# B&R Automation Studio project Ampel (part 3)

```cpp
	/// @brief Transition into a state
	///   (if transitioning into a region, activates the state that was active previously)
	/// @param `stateId` State identifier
	HFSM2_CONSTEXPR(14)	void resume   (const StateID stateId_)		noexcept;

	/// @brief Transition into a state
	///   (if transitioning into a region, activates the state that was active previously)
	/// @tparam `TState` State type
	template <typename TState>
	HFSM2_CONSTEXPR(14)	void resume   ()							noexcept	{ resume   (PlanControl::template stateId<TState>());	}

	/// @brief Transition into a state
	///   (if transitioning into a region, activates the sub-state by index returned by the region's `select()` method)
	/// @param `stateId` State identifier
	HFSM2_CONSTEXPR(14)	void select   (const StateID stateId_)		noexcept;

	/// @brief Transition into a state
	///   (if transitioning into a region, activates the sub-state by index returned by the region's `select()` method)
	/// @tparam `TState` State type
	template <typename TState>
	HFSM2_CONSTEXPR(14)	void select   ()							noexcept	{ select   (PlanControl::template stateId<TState>());	}

#if HFSM2_UTILITY_THEORY_AVAILABLE()

	/// @brief Transition into a state
	///   (if transitioning into a region, activates the state with the highest `utility()`
	///   among those with the highest `rank()`)
	/// @param `stateId` State identifier
	/// @see `HFSM2_ENABLE_UTILITY_THEORY`
	HFSM2_CONSTEXPR(14)	void utilize  (const StateID stateId_)		noexcept;

	/// @brief Transition into a state
	///   (if transitioning into a region, activates the state with the highest `utility()`
	///   among those with the highest `rank()`)
	/// @tparam `TState` State type
	/// @see `HFSM2_ENABLE_UTILITY_THEORY`
	template <typename TState>
	HFSM2_CONSTEXPR(14)	void utilize  ()							noexcept	{ utilize  (PlanControl::template stateId<TState>());	}

	/// @brief Transition into a state
	///   (if transitioning into a region, uses weighted random to activate the state proportional to `utility()`
	///   among those with the highest `rank()`)
	/// @param `stateId` State identifier
	/// @see `HFSM2_ENABLE_UTILITY_THEORY`
	HFSM2_CONSTEXPR(14)	void randomize(const StateID stateId_)		noexcept;

	/// @brief Transition into a state
	///   (if transitioning into a region, uses weighted random to activate the state proportional to `utility()`
	///   among those with the highest `rank()`)
	/// @tparam `TState` State type
	/// @see `HFSM2_ENABLE_UTILITY_THEORY`
	template <typename TState>
	HFSM2_CONSTEXPR(14)	void randomize()							noexcept	{ randomize(PlanControl::template stateId<TState>());	}

#endif

	/// @brief Schedule a state to be activated when its parent region is activated
	/// @param `stateId` State identifier
	HFSM2_CONSTEXPR(14)	void schedule (const StateID stateId_)		noexcept;

	/// @brief Schedule a state to be activated when its parent region is activated
	/// @tparam `TState` State type
	template <typename TState>
	HFSM2_CONSTEXPR(14)	void schedule ()							noexcept	{ schedule (PlanControl::template stateId<TState>());	}

#if HFSM2_PLANS_AVAILABLE()

	/// @brief Succeed a plan task for the current state
	/// @see `HFSM2_ENABLE_PLANS`
	HFSM2_CONSTEXPR(14)	void succeed()								noexcept	{ succeed  (_originId							   );	}

	/// @brief Succeed a plan task for a state
	/// @param `stateId` State identifier
	/// @see `HFSM2_ENABLE_PLANS`
	HFSM2_CONSTEXPR(14) void succeed(const StateID stateId_)		noexcept;

	/// @brief Succeed a plan task for a state
	/// @tparam `TState` State type
	/// @see `HFSM2_ENABLE_PLANS`
	template <typename TState>
	HFSM2_CONSTEXPR(14) void succeed()								noexcept	{ succeed  (PlanControl::template stateId<TState>());	}

	/// @brief Fail a plan task for the current state
	/// @see `HFSM2_ENABLE_PLANS`
	HFSM2_CONSTEXPR(14)	void fail	()								noexcept	{ fail	   (_originId							   );	}

	/// @brief Fail a plan task for a state
	/// @param `stateId` State identifier
	/// @see `HFSM2_ENABLE_PLANS`
	HFSM2_CONSTEXPR(14) void fail	(const StateID stateId_)		noexcept;

	/// @brief Fail a plan task for a state
	/// @tparam `TState` State type
	/// @see `HFSM2_ENABLE_PLANS`
	template <typename TState>
	HFSM2_CONSTEXPR(14) void fail	()								noexcept	{ fail	   (PlanControl::template stateId<TState>());	}

#endif

protected:
	using PlanControl::_core;
using PlanControl::_originId;
using PlanControl::_regionId;

using PlanControl::_regionStateId;
using PlanControl::_regionSize;
using PlanControl::_taskStatus;

bool _locked = false;
};

template <typename TArgs>
class FullControlT;

template <
	typename TConfig
  , typename TStateList
  , typename TRegionList
  , Long NCompoCount
  , Long NOrthoCount
  , Long NOrthoUnits
  , typename TReactOrder
  HFSM2_IF_SERIALIZATION(, Long NSerialBits)
  HFSM2_IF_PLANS(, Long NTaskCapacity)
  , typename TPayload
>
class FullControlT<
		  ArgsT<
			  TConfig
			, TStateList
			, TRegionList
			, NCompoCount
			, NOrthoCount
			, NOrthoUnits
			, TReactOrder
			HFSM2_IF_SERIALIZATION(, NSerialBits)
			HFSM2_IF_PLANS(, NTaskCapacity)
			, TPayload
		  >
	  >
	: public FullControlBaseT<
				 ArgsT<
					 TConfig
				   , TStateList
				   , TRegionList
				   , NCompoCount
				   , NOrthoCount
				   , NOrthoUnits
				   , TReactOrder
				   HFSM2_IF_SERIALIZATION(, NSerialBits)
				   HFSM2_IF_PLANS(, NTaskCapacity)
				   , TPayload
				 >
			 >
{
	template <typename, typename, typename>
	friend struct S_;

	template <typename, typename, Strategy, typename, typename...>
	friend struct C_;

	template <typename, typename, typename, typename...>
	friend struct O_;

	template <typename, typename>
	friend class R_;

	using Args = ArgsT<
	TConfig
	, TStateList
	, TRegionList
	, NCompoCount
	, NOrthoCount
	, NOrthoUnits
	, TReactOrder
				   HFSM2_IF_SERIALIZATION(, NSerialBits)
				   HFSM2_IF_PLANS(, NTaskCapacity)
				   , TPayload
				 >;

protected:
	using FullControlBase = FullControlBaseT<Args>;

using typename FullControlBase::Payload;
	using typename FullControlBase::Transition;

	using typename FullControlBase::Origin;

#if HFSM2_PLANS_AVAILABLE()
	using typename FullControlBase::Plan;
	using typename FullControlBase::TasksBits;
#endif

	using FullControlBase::FullControlBase;

#if HFSM2_PLANS_AVAILABLE()

	template <typename TState>
	HFSM2_CONSTEXPR(14)	TaskStatus updatePlan(TState& headState,
											  const TaskStatus subStatus)	noexcept;

#endif

public:
	using FullControlBase::context;

using FullControlBase::isActive;
using FullControlBase::changeTo;

	HFSM2_IF_PLANS(using FullControlBase::plan);

	/// @brief Transition into a state
	///   (if transitioning into a region, acts depending on the region type)
	/// @param `stateId` Destination state identifier
	/// @param `payload` Payload
	HFSM2_CONSTEXPR(14)	void changeWith   (const StateID  stateId_,
										   const Payload& payload)			noexcept;

	/// @brief Transition into a state
	///   (if transitioning into a region, acts depending on the region type)
	/// @tparam `TState` Destination state type
	/// @param `payload` Payload
	template <typename TState>
	HFSM2_CONSTEXPR(14)	void changeWith   (const Payload& payload)			noexcept	{ changeWith   (FullControlBase::template stateId<TState>(),	  payload );	}

	/// @brief Transition into a state
	///   (if transitioning into a region, activates the initial state)
	/// @param `stateId` Destination state identifier
	/// @param `payload` Payload
	HFSM2_CONSTEXPR(14)	void restartWith  (const StateID  stateId_,
										   const Payload& payload)			noexcept;

	/// @brief Transition into a state
	///   (if transitioning into a region, activates the initial state)
	/// @tparam `TState` Destination state type
	/// @param `payload` Payload
	template <typename TState>
	HFSM2_CONSTEXPR(14)	void restartWith  (const Payload& payload)			noexcept	{ restartWith  (FullControlBase::template stateId<TState>(),	  payload );	}

	/// @brief Transition into a state
	///   (if transitioning into a region, activates the state that was active previously)
	/// @param `stateId` Destination state identifier
	/// @param `payload` Payload
	HFSM2_CONSTEXPR(14)	void resumeWith   (const StateID  stateId_,
										   const Payload& payload)			noexcept;

	/// @brief Transition into a state
	///   (if transitioning into a region, activates the state that was active previously)
	/// @tparam `TState` Destination state type
	/// @param `payload` Payload
	template <typename TState>
	HFSM2_CONSTEXPR(14)	void resumeWith   (const Payload& payload)			noexcept	{ resumeWith   (FullControlBase::template stateId<TState>(),	  payload );	}

	/// @brief Transition into a state
	///   (if transitioning into a region, activates the sub-state by index returned by the region's `select()` method)
	/// @param `stateId` Destination state identifier
	/// @param `payload` Payload
	HFSM2_CONSTEXPR(14)	void selectWith   (const StateID  stateId_,
										   const Payload& payload)			noexcept;

	/// @brief Transition into a state
	///   (if transitioning into a region, activates the sub-state by index returned by the region's `select()` method)
	/// @tparam `TState` Destination state type
	/// @param `payload` Payload
	template <typename TState>
	HFSM2_CONSTEXPR(14)	void selectWith   (const Payload& payload)			noexcept	{ selectWith   (FullControlBase::template stateId<TState>(),	  payload );	}

#if HFSM2_UTILITY_THEORY_AVAILABLE()

	/// @brief Transition into a state
	///   (if transitioning into a region, activates the state with the highest `utility()`
	///   among those with the highest `rank()`)
	/// @param `stateId` Destination state identifier
	/// @param `payload` Payload
	/// @see `HFSM2_ENABLE_UTILITY_THEORY`
	HFSM2_CONSTEXPR(14)	void utilizeWith  (const StateID  stateId_,
										   const Payload& payload)			noexcept;

	/// @brief Transition into a state
	///   (if transitioning into a region, activates the state with the highest `utility()`
	///   among those with the highest `rank()`)
	/// @tparam `TState` Destination state type
	/// @param `payload` Payload
	/// @see `HFSM2_ENABLE_UTILITY_THEORY`
	template <typename TState>
	HFSM2_CONSTEXPR(14)	void utilizeWith  (const Payload& payload)			noexcept	{ utilizeWith  (FullControlBase::template stateId<TState>(),	  payload );	}

	/// @brief Transition into a state (if transitioning into a region, uses weighted random to activate the state
	///   proportional to `utility()` among those with the highest `rank()`)
	/// @param `stateId` Destination state identifier
	/// @param `payload` Payload
	/// @see `HFSM2_ENABLE_UTILITY_THEORY`
	HFSM2_CONSTEXPR(14)	void randomizeWith(const StateID  stateId_,
										   const Payload& payload)			noexcept;

	/// @brief Transition into a state (if transitioning into a region, uses weighted random to activate the state
	///   proportional to `utility()` among those with the highest `rank()`)
	/// @tparam `TState` Destination state type
	/// @param `payload` Payload
	/// @see `HFSM2_ENABLE_UTILITY_THEORY`
	template <typename TState>
	HFSM2_CONSTEXPR(14)	void randomizeWith(const Payload& payload)			noexcept	{ randomizeWith(FullControlBase::template stateId<TState>(),	  payload );	}

#endif

	/// @brief Schedule a state to be activated when its parent region is activated
	/// @param `stateId` Destination state identifier
	/// @param `payload` Payload
	HFSM2_CONSTEXPR(14)	void scheduleWith (const StateID  stateId_,
										   const Payload& payload)			noexcept;

	/// @brief Schedule a state to be activated when its parent region is activated
	/// @tparam `TState` Destination state type
	/// @param `payload` Payload
	template <typename TState>
	HFSM2_CONSTEXPR(14)	void scheduleWith (const Payload& payload)			noexcept	{ scheduleWith (FullControlBase::template stateId<TState>(),	  payload );	}

protected:
	using FullControlBase::_core;
using FullControlBase::_originId;
using FullControlBase::_regionId;

using FullControlBase::_regionStateId;
using FullControlBase::_regionSize;
using FullControlBase::_taskStatus;

using FullControlBase::_locked;
};

template <
	typename TConfig
  , typename TStateList
  , typename TRegionList
  , Long NCompoCount
  , Long NOrthoCount
  , Long NOrthoUnits
  , typename TReactOrder
  HFSM2_IF_SERIALIZATION(, Long NSerialBits)
  HFSM2_IF_PLANS(, Long NTaskCapacity)
>
class FullControlT<
		  ArgsT<
			  TConfig
			, TStateList
			, TRegionList
			, NCompoCount
			, NOrthoCount
			, NOrthoUnits
			, TReactOrder
			HFSM2_IF_SERIALIZATION(, NSerialBits)
			HFSM2_IF_PLANS(, NTaskCapacity)
			, void
		  >
	  >
	: public FullControlBaseT<
				 ArgsT<
					 TConfig
				   , TStateList
				   , TRegionList
				   , NCompoCount
				   , NOrthoCount
				   , NOrthoUnits
				   , TReactOrder
				   HFSM2_IF_SERIALIZATION(, NSerialBits)
				   HFSM2_IF_PLANS(, NTaskCapacity)
				   , void
				 >
			 >
{
	template <typename, typename, typename>
	friend struct S_;

	template <typename, typename, Strategy, typename, typename...>
	friend struct C_;

	template <typename, typename, typename, typename...>
	friend struct O_;

	template <typename, typename>
	friend class R_;

	using Args = ArgsT<
	TConfig
	, TStateList
	, TRegionList
	, NCompoCount
	, NOrthoCount
	, NOrthoUnits
	, TReactOrder
				   HFSM2_IF_SERIALIZATION(, NSerialBits)
				   HFSM2_IF_PLANS(, NTaskCapacity)
				   , void
				 >;

protected:
	using FullControlBase = FullControlBaseT<Args>;

using typename FullControlBase::Origin;

#if HFSM2_PLANS_AVAILABLE()
	using typename FullControlBase::Plan;
	using typename FullControlBase::TasksBits;
#endif

	using FullControlBase::FullControlBase;

#if HFSM2_PLANS_AVAILABLE()

	template <typename TState>
	HFSM2_CONSTEXPR(14)	TaskStatus updatePlan(TState& headState,
											  const TaskStatus subStatus)	noexcept;

#endif

public:
	using FullControlBase::context;

using FullControlBase::isActive;
using FullControlBase::changeTo;

	HFSM2_IF_PLANS(using FullControlBase::plan);

protected:
	using FullControlBase::_core;
using FullControlBase::_regionId;

using FullControlBase::_regionStateId;
using FullControlBase::_taskStatus;
};

}
}

namespace hfsm2 {
	namespace detail {

		template <typename TArgs>
		HFSM2_CONSTEXPR(14)
		FullControlBaseT<TArgs>::Lock::Lock(FullControlBaseT& control_) noexcept
	: control{!control_._locked ? &control_ : nullptr}
	{
	if (control)
	control->_locked = true;
}

template <typename TArgs>
HFSM2_CONSTEXPR(20)
FullControlBaseT<TArgs>::Lock::~Lock() noexcept {
	if (control)
control->_locked = false;
}

template <typename TArgs>
HFSM2_CONSTEXPR(14)
void
FullControlBaseT<TArgs>::changeTo(const StateID stateId_) noexcept {
	if (!_locked) {
_core.requests.emplace(Transition{_originId, stateId_, TransitionType::CHANGE});

		if (stateId_ < _regionStateId || _regionStateId + _regionSize <= stateId_)
_taskStatus.outerTransition = true;

		HFSM2_LOG_TRANSITION(context(), _originId, TransitionType::CHANGE, stateId_);
	}
}

template <typename TArgs>
HFSM2_CONSTEXPR(14)
void
FullControlBaseT<TArgs>::restart(const StateID stateId_) noexcept {
	if (!_locked) {
_core.requests.emplace(Transition{_originId, stateId_, TransitionType::RESTART});

		if (stateId_ < _regionStateId || _regionStateId + _regionSize <= stateId_)
_taskStatus.outerTransition = true;

		HFSM2_LOG_TRANSITION(context(), _originId, TransitionType::RESTART, stateId_);
	}
}

template <typename TArgs>
HFSM2_CONSTEXPR(14)
void
FullControlBaseT<TArgs>::resume(const StateID stateId_) noexcept {
	if (!_locked) {
_core.requests.emplace(Transition{_originId, stateId_, TransitionType::RESUME});

		if (stateId_ < _regionStateId || _regionStateId + _regionSize <= stateId_)
_taskStatus.outerTransition = true;

		HFSM2_LOG_TRANSITION(context(), _originId, TransitionType::RESUME, stateId_);
	}
}

template <typename TArgs>
HFSM2_CONSTEXPR(14)
void
FullControlBaseT<TArgs>::select(const StateID stateId_) noexcept {
	if (!_locked) {
_core.requests.emplace(Transition{_originId, stateId_, TransitionType::SELECT});

		if (stateId_ < _regionStateId || _regionStateId + _regionSize <= stateId_)
_taskStatus.outerTransition = true;

		HFSM2_LOG_TRANSITION(context(), _originId, TransitionType::SELECT, stateId_);
	}
}

#if HFSM2_UTILITY_THEORY_AVAILABLE()

template <typename TArgs>
HFSM2_CONSTEXPR(14)
void
FullControlBaseT<TArgs>::utilize(const StateID stateId_) noexcept {
	if (!_locked) {
		_core.requests.emplace(Transition{_originId, stateId_, TransitionType::UTILIZE});

		if (stateId_ < _regionStateId || _regionStateId + _regionSize <= stateId_)
			_taskStatus.outerTransition = true;

		HFSM2_LOG_TRANSITION(context(), _originId, TransitionType::UTILIZE, stateId_);
	}
}

template <typename TArgs>
HFSM2_CONSTEXPR(14)
void
FullControlBaseT<TArgs>::randomize(const StateID stateId_) noexcept {
	if (!_locked) {
_core.requests.emplace(Transition{_originId, stateId_, TransitionType::RANDOMIZE});

		if (stateId_ < _regionStateId || _regionStateId + _regionSize <= stateId_)
_taskStatus.outerTransition = true;

		HFSM2_LOG_TRANSITION(context(), _originId, TransitionType::RANDOMIZE, stateId_);
	}
}

#endif

template <typename TArgs>
HFSM2_CONSTEXPR(14)
void
FullControlBaseT<TArgs>::schedule(const StateID stateId_) noexcept {
_core.requests.emplace(Transition{_originId, stateId_, TransitionType::SCHEDULE});

	HFSM2_LOG_TRANSITION(context(), _originId, TransitionType::SCHEDULE, stateId_);
}

#if HFSM2_PLANS_AVAILABLE()

template <typename TArgs>
HFSM2_CONSTEXPR(14)
void
FullControlBaseT<TArgs>::succeed(const StateID stateId_) noexcept {
	if (ROOT_ID < stateId_ && stateId_ < STATE_COUNT) {
_taskStatus.result = TaskStatus::SUCCESS;

		_core.planData.tasksSuccesses.set(stateId_);

		HFSM2_LOG_TASK_STATUS(context(), _regionStateId, stateId_, StatusEvent::SUCCEEDED);
	}
}

template <typename TArgs>
HFSM2_CONSTEXPR(14)
void
FullControlBaseT<TArgs>::fail(const StateID stateId_) noexcept {
	if (ROOT_ID < stateId_ && stateId_ < STATE_COUNT) {
_taskStatus.result = TaskStatus::FAILURE;

		_core.planData.tasksFailures.set(stateId_);

		HFSM2_LOG_TASK_STATUS(context(), _regionStateId, stateId_, StatusEvent::FAILED);
	}
}

#endif

#if HFSM2_PLANS_AVAILABLE()

template <typename TG_, typename TSL_, typename TRL_, Long NCC_, Long NOC_, Long NOU_, typename TRO_ HFSM2_IF_SERIALIZATION(, Long NSB_), Long NTC_, typename TTP_>
template <typename TState>
HFSM2_CONSTEXPR(14)
TaskStatus
	FullControlT<ArgsT<TG_, TSL_, TRL_, NCC_, NOC_, NOU_, TRO_ HFSM2_IF_SERIALIZATION(, NSB_), NTC_, TTP_>>::updatePlan(TState& headState,
																													const TaskStatus subStatus) noexcept
{
constexpr StateID STATE_ID = TState::STATE_ID; // SPECIFIC

	HFSM2_ASSERT(subStatus);

	if (subStatus.result == TaskStatus::FAILURE) {
_taskStatus.result = TaskStatus::FAILURE;
		HFSM2_LOG_PLAN_STATUS(context(), _regionStateId, StatusEvent::FAILED);

		headState.wrapPlanFailed(*this);

		return TaskStatus{_taskStatus.result};
	} else if (subStatus.result == TaskStatus::SUCCESS) {
if (Plan p = plan(_regionId)) {
TasksBits successesToClear;
			successesToClear.set();

for (auto it = p.begin();
				 it && isActive(it->origin);
				 ++it)
			{
				if (_core.planData.tasksSuccesses.get(it->origin)) {
Origin origin{*this, STATE_ID}; // SPECIFIC

if (const Payload* const payload = it->payload())
						changeWith(it->destination, *it->payload());
					else
						changeTo  (it->destination);

					if (it->cyclic())
						_core.planData.tasksSuccesses.clear(it->origin); // SPECIFIC
					else
						successesToClear.clear(it->origin);

					it.remove();
				}
			}

_core.planData.tasksSuccesses &= successesToClear;

			return TaskStatus{};
		} else {
_taskStatus.result = TaskStatus::SUCCESS;
			HFSM2_LOG_PLAN_STATUS(context(), _regionStateId, StatusEvent::SUCCEEDED);

			plan().clearTasks();
			headState.wrapPlanSucceeded(*this);

			return TaskStatus{_taskStatus.result};
		}
	} else
		return TaskStatus{};
}

#endif

template <typename TG_, typename TSL_, typename TRL_, Long NCC_, Long NOC_, Long NOU_, typename TRO_ HFSM2_IF_SERIALIZATION(, Long NSB_) HFSM2_IF_PLANS(, Long NTC_), typename TTP_>
HFSM2_CONSTEXPR(14)
void
FullControlT<ArgsT<TG_, TSL_, TRL_, NCC_, NOC_, NOU_, TRO_ HFSM2_IF_SERIALIZATION(, NSB_) HFSM2_IF_PLANS(, NTC_), TTP_>>::changeWith(const StateID  stateId_,
																																	 const Payload& payload) noexcept
{
	if (!_locked) {
_core.requests.emplace(Transition{_originId, stateId_, TransitionType::CHANGE, payload});

		if (stateId_ < _regionStateId || _regionStateId + _regionSize <= stateId_)
_taskStatus.outerTransition = true;

		HFSM2_LOG_TRANSITION(context(), _originId, TransitionType::CHANGE, stateId_);
	}
}

template <typename TG_, typename TSL_, typename TRL_, Long NCC_, Long NOC_, Long NOU_, typename TRO_ HFSM2_IF_SERIALIZATION(, Long NSB_) HFSM2_IF_PLANS(, Long NTC_), typename TTP_>
HFSM2_CONSTEXPR(14)
void
FullControlT<ArgsT<TG_, TSL_, TRL_, NCC_, NOC_, NOU_, TRO_ HFSM2_IF_SERIALIZATION(, NSB_) HFSM2_IF_PLANS(, NTC_), TTP_>>::restartWith(const StateID  stateId_,
																																	  const Payload& payload) noexcept
{
	if (!_locked) {
_core.requests.emplace(Transition{_originId, stateId_, TransitionType::RESTART, payload});

		if (stateId_ < _regionStateId || _regionStateId + _regionSize <= stateId_)
_taskStatus.outerTransition = true;

		HFSM2_LOG_TRANSITION(context(), _originId, TransitionType::RESTART, stateId_);
	}
}

template <typename TG_, typename TSL_, typename TRL_, Long NCC_, Long NOC_, Long NOU_, typename TRO_ HFSM2_IF_SERIALIZATION(, Long NSB_) HFSM2_IF_PLANS(, Long NTC_), typename TTP_>
HFSM2_CONSTEXPR(14)
void
FullControlT<ArgsT<TG_, TSL_, TRL_, NCC_, NOC_, NOU_, TRO_ HFSM2_IF_SERIALIZATION(, NSB_) HFSM2_IF_PLANS(, NTC_), TTP_>>::resumeWith(const StateID  stateId_,
																																	 const Payload& payload) noexcept
{
	if (!_locked) {
_core.requests.emplace(Transition{_originId, stateId_, TransitionType::RESUME, payload});

		if (stateId_ < _regionStateId || _regionStateId + _regionSize <= stateId_)
_taskStatus.outerTransition = true;

		HFSM2_LOG_TRANSITION(context(), _originId, TransitionType::RESUME, stateId_);
	}
}

template <typename TG_, typename TSL_, typename TRL_, Long NCC_, Long NOC_, Long NOU_, typename TRO_ HFSM2_IF_SERIALIZATION(, Long NSB_) HFSM2_IF_PLANS(, Long NTC_), typename TTP_>
HFSM2_CONSTEXPR(14)
void
FullControlT<ArgsT<TG_, TSL_, TRL_, NCC_, NOC_, NOU_, TRO_ HFSM2_IF_SERIALIZATION(, NSB_) HFSM2_IF_PLANS(, NTC_), TTP_>>::selectWith(const StateID  stateId_,
																																	 const Payload& payload) noexcept
{
	if (!_locked) {
_core.requests.emplace(Transition{_originId, stateId_, TransitionType::SELECT, payload});

		if (stateId_ < _regionStateId || _regionStateId + _regionSize <= stateId_)
_taskStatus.outerTransition = true;

		HFSM2_LOG_TRANSITION(context(), _originId, TransitionType::SELECT, stateId_);
	}
}

#if HFSM2_UTILITY_THEORY_AVAILABLE()

template <typename TG_, typename TSL_, typename TRL_, Long NCC_, Long NOC_, Long NOU_, typename TRO_ HFSM2_IF_SERIALIZATION(, Long NSB_) HFSM2_IF_PLANS(, Long NTC_), typename TTP_>
HFSM2_CONSTEXPR(14)
void
FullControlT<ArgsT<TG_, TSL_, TRL_, NCC_, NOC_, NOU_, TRO_ HFSM2_IF_SERIALIZATION(, NSB_) HFSM2_IF_PLANS(, NTC_), TTP_>>::utilizeWith(const StateID  stateId_,
																																	  const Payload& payload) noexcept
{
	if (!_locked) {
		_core.requests.emplace(Transition{_originId, stateId_, TransitionType::UTILIZE, payload});

		if (stateId_ < _regionStateId || _regionStateId + _regionSize <= stateId_)
			_taskStatus.outerTransition = true;

		HFSM2_LOG_TRANSITION(context(), _originId, TransitionType::UTILIZE, stateId_);
	}
}

template <typename TG_, typename TSL_, typename TRL_, Long NCC_, Long NOC_, Long NOU_, typename TRO_ HFSM2_IF_SERIALIZATION(, Long NSB_) HFSM2_IF_PLANS(, Long NTC_), typename TTP_>
HFSM2_CONSTEXPR(14)
void
FullControlT<ArgsT<TG_, TSL_, TRL_, NCC_, NOC_, NOU_, TRO_ HFSM2_IF_SERIALIZATION(, NSB_) HFSM2_IF_PLANS(, NTC_), TTP_>>::randomizeWith(const StateID  stateId_,
																																		const Payload& payload) noexcept
{
	if (!_locked) {
		_core.requests.emplace(Transition{_originId, stateId_, TransitionType::RANDOMIZE, payload});

		if (stateId_ < _regionStateId || _regionStateId + _regionSize <= stateId_)
			_taskStatus.outerTransition = true;

		HFSM2_LOG_TRANSITION(context(), _originId, TransitionType::RANDOMIZE, stateId_);
	}
}

#endif

template <typename TG_, typename TSL_, typename TRL_, Long NCC_, Long NOC_, Long NOU_, typename TRO_ HFSM2_IF_SERIALIZATION(, Long NSB_) HFSM2_IF_PLANS(, Long NTC_), typename TTP_>
HFSM2_CONSTEXPR(14)
void
FullControlT<ArgsT<TG_, TSL_, TRL_, NCC_, NOC_, NOU_, TRO_ HFSM2_IF_SERIALIZATION(, NSB_) HFSM2_IF_PLANS(, NTC_), TTP_>>::scheduleWith(const StateID  stateId_,
																																	   const Payload& payload) noexcept
{
_core.requests.emplace(Transition{_originId, stateId_, TransitionType::SCHEDULE, payload});

	HFSM2_LOG_TRANSITION(context(), _originId, TransitionType::SCHEDULE, stateId_);
}

#if HFSM2_PLANS_AVAILABLE()

template <typename TG_, typename TSL_, typename TRL_, Long NCC_, Long NOC_, Long NOU_, typename TRO_ HFSM2_IF_SERIALIZATION(, Long NSB_), Long NTC_>
template <typename TState>
HFSM2_CONSTEXPR(14)
TaskStatus
FullControlT<ArgsT<TG_, TSL_, TRL_, NCC_, NOC_, NOU_, TRO_ HFSM2_IF_SERIALIZATION(, NSB_), NTC_, void>>::updatePlan(TState& headState,
																													const TaskStatus subStatus) noexcept
{
constexpr StateID STATE_ID = TState::STATE_ID; // SPECIFIC

	HFSM2_ASSERT(subStatus);

	if (subStatus.result == TaskStatus::FAILURE) {
_taskStatus.result = TaskStatus::FAILURE;
		HFSM2_LOG_PLAN_STATUS(context(), _regionStateId, StatusEvent::FAILED);

		headState.wrapPlanFailed(*this);

		return TaskStatus{_taskStatus.result};
	} else if (subStatus.result == TaskStatus::SUCCESS) {
if (Plan p = plan(_regionId)) {
TasksBits successesToClear;
			successesToClear.set();

for (auto it = p.begin();
				 it && isActive(it->origin);
				 ++it)
			{
				if (_core.planData.tasksSuccesses.get(it->origin)) {
Origin origin{*this, STATE_ID}; // SPECIFIC

					changeTo(it->destination);

					if (it->cyclic())
						_core.planData.tasksSuccesses.clear(it->origin); // SPECIFIC
					else
						successesToClear.clear(it->origin);

					it.remove();
				}
			}

_core.planData.tasksSuccesses &= successesToClear;

			return TaskStatus{};
		} else {
_taskStatus.result = TaskStatus::SUCCESS;
			HFSM2_LOG_PLAN_STATUS(context(), _regionStateId, StatusEvent::SUCCEEDED);

			plan().clearTasks();
			headState.wrapPlanSucceeded(*this);

			return TaskStatus{_taskStatus.result};
		}
	} else
		return TaskStatus{};
}

#endif

}
}

namespace hfsm2 {
	namespace detail {

		template <typename TArgs>
		class GuardControlT final
		: public FullControlT<TArgs>
		{
		template <typename, typename, typename>
		friend struct S_;

		template <typename, typename>
		friend class R_;

		using FullControl	= FullControlT<TArgs>;

		using typename FullControl::Core;
		using typename FullControl::Context;

		using typename FullControl::Registry;
		using typename FullControl::TransitionSet;
		using typename FullControl::TransitionSets;

#if HFSM2_TRANSITION_HISTORY_AVAILABLE()
		using typename FullControl::TransitionTargets;
#endif

#if HFSM2_UTILITY_THEORY_AVAILABLE()
		using typename FullControl::RNG;
#endif

#if HFSM2_PLANS_AVAILABLE()
		using typename FullControl::PlanData;
#endif

#if HFSM2_LOG_INTERFACE_AVAILABLE()
		using typename FullControl::Logger;
#endif

		HFSM2_CONSTEXPR(11)	GuardControlT(Core& core,
		const TransitionSets& currentTransitions,
		const TransitionSet& pendingTransitions) noexcept
		: FullControl{core, currentTransitions}
, _pendingTransitions{pendingTransitions}
	{}

public:
	using FullControl::context;

	/// @brief Check if a state is going to be activated or deactivated
	/// @param `stateId` State identifier
	/// @return State pending activation/deactivation status
	HFSM2_CONSTEXPR(11)	bool isPendingChange(const StateID stateId_)  const noexcept	{ return _core.registry.isPendingChange(stateId_);					}

	/// @brief Check if a state is going to be activated or deactivated
	/// @tparam `TState` State type
	/// @return State pending activation/deactivation status
	template <typename TState>
	HFSM2_CONSTEXPR(11)	bool isPendingChange()						  const noexcept	{ return isPendingChange(FullControl::template stateId<TState>());	}

	/// @brief Check if a state is going to be activated
	/// @param `stateId` State identifier
	/// @return State pending activation status
	HFSM2_CONSTEXPR(11)	bool isPendingEnter (const StateID stateId_)  const noexcept	{ return _core.registry.isPendingEnter (stateId_);					}

	/// @brief Check if a state is going to be activated
	/// @tparam `TState` State type
	/// @return State pending activation status
	template <typename TState>
	HFSM2_CONSTEXPR(11)	bool isPendingEnter ()						  const noexcept	{ return isPendingEnter (FullControl::template stateId<TState>());	}

	/// @brief Check if a state is going to be deactivated
	/// @param `stateId` State identifier
	/// @return State pending deactivation status
	HFSM2_CONSTEXPR(11)	bool isPendingExit	(const StateID stateId_)  const noexcept	{ return _core.registry.isPendingExit  (stateId_);					}

	/// @brief Check if a state is going to be deactivated
	/// @tparam `TState` State type
	/// @return State pending deactivation status
	template <typename TState>
	HFSM2_CONSTEXPR(11)	bool isPendingExit  ()						  const noexcept	{ return isPendingExit  (FullControl::template stateId<TState>());	}

	/// @brief Get pending transition requests
	/// @return Array of pending transition requests
	HFSM2_CONSTEXPR(11)	const TransitionSet&  pendingTransitions()	  const noexcept	{ return _pendingTransitions;										}

	/// @brief Cancel pending transition requests
	///   (can be used to substitute a transition into the current state with a different one)
	HFSM2_CONSTEXPR(14)	void cancelPendingTransitions()						noexcept;

private:
	using FullControl::_core;
using FullControl::_originId;

const TransitionSet& _pendingTransitions;

bool _cancelled = false;
};

}
}

namespace hfsm2 {
	namespace detail {

		template <typename TArgs>
		HFSM2_CONSTEXPR(14)
		void
		GuardControlT<TArgs>::cancelPendingTransitions() noexcept {
		_cancelled = true;

		HFSM2_LOG_CANCELLED_PENDING(context(), _originId);
	}

}
}

namespace hfsm2 {
	namespace detail {

		template <typename TArgs>
		class EventControlT final
		: public FullControlT<TArgs>
		{
		template <typename, typename>
		friend class R_;

		template <typename, typename>
		friend struct PreReactWrapperT;

		template <typename, typename>
		friend struct ReactWrapperT;

		template <typename, typename>
		friend struct PostReactWrapperT;

		using FullControl	= FullControlT<TArgs>;

		using FullControl::FullControl;

		public:
		using FullControl::context;

		/// @brief Stops processing of the current event down the hierarchy
		/// @see `Config::BottomUpReactions`
	HFSM2_CONSTEXPR(14)	void consumeEvent()								noexcept	{ _consumed = true;	}

	private:
	bool _consumed = false;
};

}
}

namespace hfsm2 {
	namespace detail {

		template <typename TArgs>
		class B_ {
			template <typename...>
			friend struct A_;

			protected:
			using Context		= typename TArgs::Context;

			using Short			= ::hfsm2::Short;
			using Prong			= ::hfsm2::Prong;

#if HFSM2_UTILITY_THEORY_AVAILABLE()
			using Rank			= typename TArgs::Rank;
			using Utility		= typename TArgs::Utility;
#endif

			using StateList		= typename TArgs::StateList;
			using RegionList	= typename TArgs::RegionList;

			using Payload		= typename TArgs::Payload;
			using Transition	= TransitionT<Payload>;

			using ConstControl	= ConstControlT<TArgs>;
			using Control		= ControlT	   <TArgs>;
			using PlanControl	= PlanControlT <TArgs>;
			using FullControl	= FullControlT <TArgs>;
			using GuardControl	= GuardControlT<TArgs>;
			using EventControl	= EventControlT<TArgs>;

#if HFSM2_PLANS_AVAILABLE()
			using Plan			= PayloadPlanT <TArgs>;
#endif

			public:

		HFSM2_CONSTEXPR(14)	void	 entryGuard	  (GuardControl&		 )			noexcept	{}

	HFSM2_CONSTEXPR(14)	void	 enter		  ( PlanControl&		 )			noexcept	{}
HFSM2_CONSTEXPR(14)	void	 reenter	  ( PlanControl&		 )			noexcept	{}

	HFSM2_CONSTEXPR(14)	void	 preUpdate	  ( FullControl&		 )			noexcept	{}
	HFSM2_CONSTEXPR(14)	void	 update		  ( FullControl&		 )			noexcept	{}
	HFSM2_CONSTEXPR(14)	void	 postUpdate	  ( FullControl&		 )			noexcept	{}

	template <typename TEvent>
	HFSM2_CONSTEXPR(14)	void	 preReact	  (const TEvent&		 ,
											   EventControl&		 )			noexcept	{}

	template <typename TEvent>
	HFSM2_CONSTEXPR(14)	void	 react		  (const TEvent&		 ,
											   EventControl&		 )			noexcept	{}

	template <typename TEvent>
	HFSM2_CONSTEXPR(14)	void	 postReact	  (const TEvent&		 ,
											   EventControl&		 )			noexcept	{}

	template <typename TEvent>
	HFSM2_CONSTEXPR(14)	void	 query		  (		 TEvent&		 ,
ConstControl&		 )	  const noexcept	{}

	HFSM2_CONSTEXPR(14)	void	 exitGuard	  (GuardControl&		 )			noexcept	{}

	HFSM2_CONSTEXPR(14)	void	 exit		  ( PlanControl&		 )			noexcept	{}

	template <typename TState>
	static
	HFSM2_CONSTEXPR(11) StateID  stateId()										noexcept	{ return					   index<StateList , TState>() ;	}

	template <typename TState>
	static
	HFSM2_CONSTEXPR(11) RegionID regionId()										noexcept	{ return static_cast<RegionID>(index<RegionList, TState>());	}
};

}
}

namespace hfsm2 {
	namespace detail {

		template <typename...>
		struct A_;

		template <typename TArgs>
		using EmptyT = A_<B_<TArgs>>;

		template <typename TFirst, typename... TRest>
		struct HFSM2_EMPTY_BASES A_<TFirst, TRest...>
		: TFirst
		, A_<TRest...>
		{
		using First		= TFirst;
		using typename First::Context;

#if HFSM2_UTILITY_THEORY_AVAILABLE()
		using typename First::Rank;
		using typename First::Utility;
#endif

		using typename First::StateList;
		using typename First::RegionList;

		using typename First::ConstControl;
		using typename First::Control;
		using typename First::PlanControl;

#if HFSM2_PLANS_AVAILABLE()
		using typename First::Plan;
#endif

		using typename First::FullControl;
		using typename First::GuardControl;
		using typename First::EventControl;

		using First::stateId;
		using First::regionId;

		using Rest		= A_<TRest...>;

		HFSM2_CONSTEXPR(14)	void	 wideEntryGuard(GuardControl& control)			noexcept;

		HFSM2_CONSTEXPR(14)	void	 wideEnter	   ( PlanControl& control)			noexcept;
		HFSM2_CONSTEXPR(14)	void	 wideReenter   ( PlanControl& control)			noexcept;

		HFSM2_CONSTEXPR(14)	void	 widePreUpdate ( FullControl& control)			noexcept;
		HFSM2_CONSTEXPR(14)	void	 wideUpdate	   ( FullControl& control)			noexcept;
		HFSM2_CONSTEXPR(14)	void	 widePostUpdate( FullControl& control)			noexcept;

		template <typename TEvent>
		HFSM2_CONSTEXPR(14)	void	 widePreReact  (const TEvent& event	 ,
		EventControl& control)			noexcept;

		template <typename TEvent>
		HFSM2_CONSTEXPR(14)	void	 wideReact	   (const TEvent& event	 ,
		EventControl& control)			noexcept;

		template <typename TEvent>
		HFSM2_CONSTEXPR(14)	void	 widePostReact (const TEvent& event	 ,
		EventControl& control)			noexcept;

		template <typename TEvent>
		HFSM2_CONSTEXPR(14)	void	 wideQuery	   (	  TEvent& event	 ,
		ConstControl& control)	  const noexcept;

		HFSM2_CONSTEXPR(14)	void	 wideExitGuard (GuardControl& control)			noexcept;

		HFSM2_CONSTEXPR(14)	void	 wideExit	   ( PlanControl& control)			noexcept;

	};

}
}

namespace hfsm2 {
	namespace detail {

		template <typename TF_, typename... TR_>
		HFSM2_CONSTEXPR(14)
		void
		A_<TF_, TR_...>::wideEntryGuard(GuardControl& control) noexcept {
		First::	   entryGuard(control);
		Rest ::wideEntryGuard(control);
	}

	template <typename TF_, typename... TR_>
	HFSM2_CONSTEXPR(14)
	void
	A_<TF_, TR_...>::wideEnter(PlanControl& control) noexcept {
	First::	   enter(control);
	Rest ::wideEnter(control);
}

template <typename TF_, typename... TR_>
HFSM2_CONSTEXPR(14)
void
A_<TF_, TR_...>::wideReenter(PlanControl& control) noexcept {
	First::	   reenter(control);
	Rest ::wideReenter(control);
}

template <typename TF_, typename... TR_>
HFSM2_CONSTEXPR(14)
void
A_<TF_, TR_...>::widePreUpdate(FullControl& control) noexcept {
	First::	   preUpdate(control);
	Rest ::widePreUpdate(control);
}

template <typename TF_, typename... TR_>
HFSM2_CONSTEXPR(14)
void
A_<TF_, TR_...>::wideUpdate(FullControl& control) noexcept {
	First::	   update(control);
	Rest ::wideUpdate(control);
}

template <typename TF_, typename... TR_>
HFSM2_CONSTEXPR(14)
void
A_<TF_, TR_...>::widePostUpdate(FullControl& control) noexcept {
	Rest ::widePostUpdate(control);
	First::	   postUpdate(control);
}

template <typename TF_, typename... TR_>
template <typename TEvent>
HFSM2_CONSTEXPR(14)
void
A_<TF_, TR_...>::widePreReact(const TEvent& event,
							  EventControl& control) noexcept
{
	First::	   preReact(event, control);
	Rest ::widePreReact(event, control);
}

template <typename TF_, typename... TR_>
template <typename TEvent>
HFSM2_CONSTEXPR(14)
void
A_<TF_, TR_...>::wideReact(const TEvent& event,
						   EventControl& control) noexcept
{
	First::	   react(event, control);
	Rest ::wideReact(event, control);
}

template <typename TF_, typename... TR_>
template <typename TEvent>
HFSM2_CONSTEXPR(14)
void
A_<TF_, TR_...>::widePostReact(const TEvent& event,
							   EventControl& control) noexcept
{
	Rest ::widePostReact(event, control);
	First::	   postReact(event, control);
}

template <typename TF_, typename... TR_>
template <typename TEvent>
HFSM2_CONSTEXPR(14)
void
A_<TF_, TR_...>::wideQuery(TEvent& event,
						   ConstControl& control) const noexcept
{
	First::	   query(event, control);
	Rest ::wideQuery(event, control);
}

template <typename TF_, typename... TR_>
HFSM2_CONSTEXPR(14)
void
A_<TF_, TR_...>::wideExitGuard(GuardControl& control) noexcept {
	Rest ::wideExitGuard(control);
	First::	   exitGuard(control);
}

template <typename TF_, typename... TR_>
HFSM2_CONSTEXPR(14)
void
A_<TF_, TR_...>::wideExit(PlanControl& control) noexcept {
	Rest ::wideExit(control);
	First::	   exit(control);
}

}
}

namespace hfsm2 {
	namespace detail {

		template <typename TFirst>
		struct HFSM2_EMPTY_BASES A_<TFirst>
			: TFirst
			{
			using First		= TFirst;
			using typename First::Context;

#if HFSM2_UTILITY_THEORY_AVAILABLE()
			using typename First::Rank;
			using typename First::Utility;
#endif

			using typename First::StateList;
			using typename First::RegionList;

			using typename First::Payload;
			using typename First::Transition;

			using typename First::ConstControl;
			using typename First::Control;
			using typename First::PlanControl;

#if HFSM2_PLANS_AVAILABLE()
			using typename First::Plan;
#endif

			using typename First::FullControl;
			using typename First::GuardControl;
			using typename First::EventControl;

			using First::stateId;
			using First::regionId;

		HFSM2_CONSTEXPR(14)	Prong	 select		   (const Control&		 )			noexcept	{ return 0;					}

#if HFSM2_UTILITY_THEORY_AVAILABLE()
	HFSM2_CONSTEXPR(14)	Rank	 rank		   (const Control&		 )			noexcept	{ return Rank   {0};		}
	HFSM2_CONSTEXPR(14)	Utility  utility	   (const Control&		 )			noexcept	{ return Utility{1};		}
#endif

	HFSM2_CONSTEXPR(14)	void	 entryGuard	   (GuardControl&		 )			noexcept	{}

	HFSM2_CONSTEXPR(14)	void	 enter		   ( PlanControl&		 )			noexcept	{}
	HFSM2_CONSTEXPR(14)	void	 reenter	   ( PlanControl&		 )			noexcept	{}

	HFSM2_CONSTEXPR(14)	void	 preUpdate	   ( FullControl&		 )			noexcept	{}
	HFSM2_CONSTEXPR(14)	void	 update		   ( FullControl&		 )			noexcept	{}
	HFSM2_CONSTEXPR(14)	void	 postUpdate	   ( FullControl&		 )			noexcept	{}

	template <typename TEvent>
	HFSM2_CONSTEXPR(14)	void	 preReact	   (const TEvent&		 ,
												EventControl&		 )			noexcept	{}

	template <typename TEvent>
	HFSM2_CONSTEXPR(14)	void	 react		   (const TEvent&		 ,
												EventControl&		 )			noexcept	{}

	template <typename TEvent>
	HFSM2_CONSTEXPR(14)	void	 postReact	   (const TEvent&		 ,
												EventControl&		 )			noexcept	{}

	template <typename TEvent>
	HFSM2_CONSTEXPR(14)	void	 query		   (	  TEvent&		 ,
ConstControl&		 )	  const noexcept	{}

	HFSM2_CONSTEXPR(14)	void	 exitGuard	   (GuardControl&		 )			noexcept	{}

	HFSM2_CONSTEXPR(14)	void	 exit		   ( PlanControl&		 )			noexcept	{}

#if HFSM2_PLANS_AVAILABLE()
	HFSM2_CONSTEXPR(14)	void	 planSucceeded ( FullControl& control)			noexcept;
	HFSM2_CONSTEXPR(14)	void	 planFailed	   ( FullControl& control)			noexcept;
#endif

	HFSM2_CONSTEXPR(14)	void	 wideEntryGuard(GuardControl& control)			noexcept;

	HFSM2_CONSTEXPR(14)	void	 wideEnter	   ( PlanControl& control)			noexcept;
	HFSM2_CONSTEXPR(14)	void	 wideReenter   ( PlanControl& control)			noexcept;

	HFSM2_CONSTEXPR(14)	void	 widePreUpdate ( FullControl& control)			noexcept;
	HFSM2_CONSTEXPR(14)	void	 wideUpdate	   ( FullControl& control)			noexcept;
	HFSM2_CONSTEXPR(14)	void	 widePostUpdate( FullControl& control)			noexcept;

	template <typename TEvent>
	HFSM2_CONSTEXPR(14)	void	 widePreReact  (const TEvent& event	 ,
												EventControl& control)			noexcept;

	template <typename TEvent>
	HFSM2_CONSTEXPR(14)	void	 wideReact	   (const TEvent& event	 ,
												EventControl& control)			noexcept;

	template <typename TEvent>
	HFSM2_CONSTEXPR(14)	void	 widePostReact (const TEvent& event	 ,
												EventControl& control)			noexcept;

	template <typename TEvent>
	HFSM2_CONSTEXPR(14)	void	 wideQuery	   (	  TEvent& event	 ,
												ConstControl& control)	  const noexcept;

	HFSM2_CONSTEXPR(14)	void	 wideExitGuard (GuardControl& control)			noexcept;

	HFSM2_CONSTEXPR(14)	void	 wideExit	   ( PlanControl& control)			noexcept;

};

}
}

namespace hfsm2 {
	namespace detail {

#if HFSM2_PLANS_AVAILABLE()

		template <typename TF_>
		HFSM2_CONSTEXPR(14)
		void
		A_<TF_>::planSucceeded(FullControl& control) noexcept {
		control.succeed();
	}

	template <typename TF_>
	HFSM2_CONSTEXPR(14)
	void
	A_<TF_>::planFailed(FullControl& control) noexcept {
	control.fail();
}

#endif

template <typename TF_>
HFSM2_CONSTEXPR(14)
void
A_<TF_>::wideEntryGuard(GuardControl& control) noexcept {
	First::	   entryGuard(control);
}

template <typename TF_>
HFSM2_CONSTEXPR(14)
void
A_<TF_>::wideEnter(PlanControl& control) noexcept {
	First::	   enter(control);
}

template <typename TF_>
HFSM2_CONSTEXPR(14)
void
A_<TF_>::wideReenter(PlanControl& control) noexcept {
	First::	   reenter(control);
}

template <typename TF_>
HFSM2_CONSTEXPR(14)
void
A_<TF_>::widePreUpdate(FullControl& control) noexcept {
	First::	   preUpdate(control);
}

template <typename TF_>
HFSM2_CONSTEXPR(14)
void
A_<TF_>::wideUpdate(FullControl& control) noexcept {
	First::	   update(control);
}

template <typename TF_>
HFSM2_CONSTEXPR(14)
void
A_<TF_>::widePostUpdate(FullControl& control) noexcept {
	First::	   postUpdate(control);
}

template <typename TF_>
template <typename TEvent>
HFSM2_CONSTEXPR(14)
void
A_<TF_>::widePreReact(const TEvent& event,
					  EventControl& control) noexcept
{
	First::	   preReact(event, control);
}

template <typename TF_>
template <typename TEvent>
HFSM2_CONSTEXPR(14)
void
A_<TF_>::wideReact(const TEvent& event,
				   EventControl& control) noexcept
{
	First::	   react(event, control);
}

template <typename TF_>
template <typename TEvent>
HFSM2_CONSTEXPR(14)
void
A_<TF_>::widePostReact(const TEvent& event,
					   EventControl& control) noexcept
{
	First::	   postReact(event, control);
}

template <typename TF_>
template <typename TEvent>
HFSM2_CONSTEXPR(14)
void
	A_<TF_>::wideQuery(TEvent& event,
	ConstControl& control) const noexcept
{
	First::	   query(event, control);
}

template <typename TF_>
HFSM2_CONSTEXPR(14)
void
A_<TF_>::wideExitGuard(GuardControl& control) noexcept {
	First::	   exitGuard(control);
}

template <typename TF_>
HFSM2_CONSTEXPR(14)
void
A_<TF_>::wideExit(PlanControl& control) noexcept {
	First::	   exit(control);
}

}
}

namespace hfsm2 {
	namespace detail {

		template <
		typename TIndices
		, typename TArgs
		, typename THead
		>
		struct HFSM2_EMPTY_BASES S_
			: THead
			{
			static constexpr StateID STATE_ID = TIndices::STATE_ID;

			using Context		= typename TArgs::Context;
			using StateList		= typename TArgs::StateList;

#if HFSM2_UTILITY_THEORY_AVAILABLE()
			using Rank			= typename TArgs::Rank;
			using Utility		= typename TArgs::Utility;
			using UP			= typename TArgs::UP;
#endif

#if HFSM2_LOG_INTERFACE_AVAILABLE()
			using Logger		= typename TArgs::Logger;
#endif

			using ConstControl	= ConstControlT<TArgs>;
			using ScopedCOrigin	= typename ConstControl::Origin;

			using Control		= ControlT	   <TArgs>;
			using Registry		= RegistryT	   <TArgs>;
			using StateParents	= typename Registry::StateParents;

			using PlanControl	= PlanControlT <TArgs>;
			using ScopedOrigin	= typename PlanControl::Origin;

			using FullControl	= FullControlT <TArgs>;
			using GuardControl	= GuardControlT<TArgs>;
			using EventControl	= EventControlT<TArgs>;

			using Empty			= EmptyT<TArgs>;
			using Head			= THead;

		HFSM2_CONSTEXPR(14)	Parent		 stateParent		  (		Control& control)								noexcept	{ return control._core.registry.stateParents[STATE_ID];	}

		HFSM2_CONSTEXPR(14)	void		 deepRegister		  (	   Registry& registry, const Parent parent)			noexcept;

		HFSM2_CONSTEXPR(14)	Prong		 wrapSelect			  (		Control& control)								noexcept;

#if HFSM2_UTILITY_THEORY_AVAILABLE()
		HFSM2_CONSTEXPR(14)	Rank		 wrapRank			  (		Control& control)								noexcept;
		HFSM2_CONSTEXPR(14)	Utility		 wrapUtility		  (		Control& control)								noexcept;
#endif

	HFSM2_CONSTEXPR(14)	bool		 deepForwardEntryGuard(GuardControl&		)								noexcept	{ return false;		}
	HFSM2_CONSTEXPR(14)	bool		 deepEntryGuard		  (GuardControl& control)								noexcept;

	HFSM2_CONSTEXPR(14)	void		 deepEnter			  ( PlanControl& control)								noexcept;
	HFSM2_CONSTEXPR(14)	void		 deepReenter		  ( PlanControl& control)								noexcept;

	HFSM2_CONSTEXPR(14)	TaskStatus	 deepPreUpdate		  ( FullControl& control)								noexcept;
	HFSM2_CONSTEXPR(14)	TaskStatus	 deepUpdate			  ( FullControl& control)								noexcept;
	HFSM2_CONSTEXPR(14)	TaskStatus	 deepPostUpdate		  ( FullControl& control)								noexcept;

	template <typename TEvent>
	HFSM2_CONSTEXPR(14)	TaskStatus	 deepPreReact		  (EventControl& control, const TEvent&	event)			noexcept;

	template <typename TEvent>
	HFSM2_CONSTEXPR(14)	TaskStatus	 deepReact			  (EventControl& control, const TEvent&	event)			noexcept;

	template <typename TEvent>
	HFSM2_CONSTEXPR(14)	TaskStatus	 deepPostReact		  (EventControl& control, const TEvent&	event)			noexcept;

	template <typename TEvent>
	HFSM2_CONSTEXPR(14)	void		 deepQuery			  (ConstControl& control,		TEvent& event)	  const noexcept;

#if HFSM2_PLANS_AVAILABLE()
	HFSM2_CONSTEXPR(14)	TaskStatus	 deepUpdatePlans	  ( FullControl& control)								noexcept;
#endif

HFSM2_CONSTEXPR(14)	bool		 deepForwardExitGuard (GuardControl&		)								noexcept	{ return false;		}
	HFSM2_CONSTEXPR(14)	bool		 deepExitGuard		  (GuardControl& control)								noexcept;

	HFSM2_CONSTEXPR(14)	void		 deepExit			  ( PlanControl& control)								noexcept;

#if HFSM2_PLANS_AVAILABLE()
	HFSM2_CONSTEXPR(14)	void		 wrapPlanSucceeded	  ( FullControl& control)								noexcept;
	HFSM2_CONSTEXPR(14)	void		 wrapPlanFailed		  ( FullControl& control)								noexcept;
#endif

	HFSM2_CONSTEXPR(14)	void		 deepForwardActive	  (	    Control&,		  const Request		   )		noexcept	{}
	HFSM2_CONSTEXPR(14)	void		 deepForwardRequest	  (	    Control& control, const Request request)		noexcept;

	HFSM2_CONSTEXPR(14)	void		 deepRequestChange	  (	    Control& control, const Request request)		noexcept;
	HFSM2_CONSTEXPR(14)	void		 deepRequestRestart	  (		Control& control, const Request request)		noexcept;
	HFSM2_CONSTEXPR(14)	void		 deepRequestResume	  (		Control& control, const Request request)		noexcept;
	HFSM2_CONSTEXPR(14)	void		 deepRequestSelect	  (	    Control& control, const Request request)		noexcept;

#if HFSM2_UTILITY_THEORY_AVAILABLE()
	HFSM2_CONSTEXPR(14)	void		 deepRequestUtilize	  (		Control& control, const Request request)		noexcept;
	HFSM2_CONSTEXPR(14)	void		 deepRequestRandomize (		Control& control, const Request request)		noexcept;

	HFSM2_CONSTEXPR(14)	UP			 deepReportChange	  (	    Control& control)								noexcept;
	HFSM2_CONSTEXPR(14)	UP			 deepReportUtilize	  (	    Control& control)								noexcept;
	HFSM2_CONSTEXPR(14)	Rank		 deepReportRank		  (		Control& control)								noexcept;
	HFSM2_CONSTEXPR(14)	Utility		 deepReportRandomize  (	    Control& control)								noexcept;
#endif

	HFSM2_CONSTEXPR(14)	void		 deepChangeToRequested(	   Control&)										noexcept	{}

#if HFSM2_SERIALIZATION_AVAILABLE()
	using WriteStream	= typename TArgs::WriteStream;
	using ReadStream	= typename TArgs::ReadStream;

	HFSM2_CONSTEXPR(14)	void		 deepSaveActive		  (const Registry&, WriteStream&)				  const noexcept	{}
	HFSM2_CONSTEXPR(14)	void		 deepSaveResumable	  (const Registry&, WriteStream&)				  const noexcept	{}

	HFSM2_CONSTEXPR(14)	void		 deepLoadRequested	  (		 Registry&,  ReadStream&)				  const noexcept	{}
	HFSM2_CONSTEXPR(14)	void		 deepLoadResumable	  (		 Registry&,  ReadStream&)				  const noexcept	{}
#endif

#if HFSM2_STRUCTURE_REPORT_AVAILABLE()
	using StructureStateInfos = typename TArgs::StructureStateInfos;

	static
	HFSM2_CONSTEXPR(NO)	const char* name() noexcept;

	HFSM2_CONSTEXPR(14)	void deepGetNames(const Long parent,
										  const RegionType region,
										  const Short depth,
										  StructureStateInfos& stateInfos)							  const noexcept;
#endif

#if HFSM2_DEBUG_STATE_TYPE_AVAILABLE() || HFSM2_STRUCTURE_REPORT_AVAILABLE() || HFSM2_LOG_INTERFACE_AVAILABLE()

	HFSM2_IF_TYPEINDEX(const std::type_index TYPE = typeid(Head));

	static constexpr Long NAME_COUNT = 1;

#endif

#if HFSM2_LOG_INTERFACE_AVAILABLE()

	template <typename TReturn, typename THost, typename... TParams>
	HFSM2_CONSTEXPR(14)
	void log(TReturn (THost::*)(TParams...),
Logger& logger,
const Context& context,
const Method method)																	  const noexcept
	{
		logger.recordMethod(context, STATE_ID, method);
	}

	template <typename TReturn, typename THost, typename... TParams>
	HFSM2_CONSTEXPR(14)
	void log(TReturn (THost::*)(TParams...) const,
Logger& logger,
const Context& context,
const Method method)																	  const noexcept
	{
		logger.recordMethod(context, STATE_ID, method);
	}

	template <typename TReturn, typename... TParams>
	HFSM2_CONSTEXPR(14)
	void log(TReturn (Empty::*)(TParams...),
Logger&,
const Context&,
			 const Method)																			  const noexcept
	{}

	template <typename TReturn, typename... TParams>
	HFSM2_CONSTEXPR(14)
	void log(TReturn (Empty::*)(TParams...) const,
Logger&,
const Context&,
			 const Method)																			  const noexcept
	{}

#endif
};

}
}

namespace hfsm2 {
	namespace detail {

		template <typename TN_, typename TA_, typename TH_>
		HFSM2_CONSTEXPR(14)
		void
		S_<TN_, TA_, TH_>::deepRegister(Registry& registry,
		const Parent parent) noexcept
		{
		constexpr StateID HEAD_ID = index<StateList, TH_>();
		static_assert(STATE_ID == HEAD_ID, "");

		registry.stateParents[STATE_ID] = parent;
	}

	template <typename TN_, typename TA_, typename TH_>
	HFSM2_CONSTEXPR(14)
	Prong
	S_<TN_, TA_, TH_>::wrapSelect(Control& control) noexcept {
	HFSM2_LOG_STATE_METHOD(&Head::select,
	Method::SELECT);

	return Head::select(static_cast<const Control&>(control));
}

#if HFSM2_UTILITY_THEORY_AVAILABLE()

template <typename TN_, typename TA_, typename TH_>
HFSM2_CONSTEXPR(14)
typename S_<TN_, TA_, TH_>::Rank
S_<TN_, TA_, TH_>::wrapRank(Control& control) noexcept {
	HFSM2_LOG_STATE_METHOD(&Head::rank,
						   Method::RANK);

	return Head::rank(static_cast<const Control&>(control));
}

template <typename TN_, typename TA_, typename TH_>
HFSM2_CONSTEXPR(14)
typename S_<TN_, TA_, TH_>::Utility
S_<TN_, TA_, TH_>::wrapUtility(Control& control) noexcept {
	HFSM2_LOG_STATE_METHOD(&Head::utility,
						   Method::UTILITY);

	return Head::utility(static_cast<const Control&>(control));
}

#endif

template <typename TN_, typename TA_, typename TH_>
HFSM2_CONSTEXPR(14)
bool
S_<TN_, TA_, TH_>::deepEntryGuard(GuardControl& control) noexcept {
	HFSM2_LOG_STATE_METHOD(&Head::entryGuard,
						   Method::ENTRY_GUARD);

ScopedOrigin origin{control, STATE_ID};

const bool cancelledBefore = control._cancelled;

	Head::wideEntryGuard(control);
	Head::	  entryGuard(control);

return !cancelledBefore && control._cancelled;
}

template <typename TN_, typename TA_, typename TH_>
HFSM2_CONSTEXPR(14)
void
S_<TN_, TA_, TH_>::deepEnter(PlanControl& control) noexcept {
	HFSM2_IF_PLANS(control._core.planData.verifyEmptyStatus(STATE_ID));

	HFSM2_LOG_STATE_METHOD(&Head::enter,
						   Method::ENTER);

ScopedOrigin origin{control, STATE_ID};

	Head::wideEnter(control);
	Head::	  enter(control);
}

template <typename TN_, typename TA_, typename TH_>
HFSM2_CONSTEXPR(14)
void
S_<TN_, TA_, TH_>::deepReenter(PlanControl& control) noexcept {
	HFSM2_IF_PLANS(control._core.planData.verifyEmptyStatus(STATE_ID));

	HFSM2_LOG_STATE_METHOD(&Head::reenter,
						   Method::REENTER);

ScopedOrigin origin{control, STATE_ID};

	Head::wideReenter(control);
	Head::	  reenter(control);
}

template <typename TN_, typename TA_, typename TH_>
HFSM2_CONSTEXPR(14)
TaskStatus
S_<TN_, TA_, TH_>::deepPreUpdate(FullControl& control) noexcept {
	HFSM2_LOG_STATE_METHOD(&Head::preUpdate,
						   Method::PRE_UPDATE);

ScopedOrigin origin{control, STATE_ID};

	Head::widePreUpdate(control);
	Head::	  preUpdate(control);

return control._taskStatus;
}

template <typename TN_, typename TA_, typename TH_>
HFSM2_CONSTEXPR(14)
TaskStatus
S_<TN_, TA_, TH_>::deepUpdate(FullControl& control) noexcept {
	HFSM2_LOG_STATE_METHOD(&Head::update,
						   Method::UPDATE);

ScopedOrigin origin{control, STATE_ID};

	Head::wideUpdate(control);
	Head::	  update(control);

return control._taskStatus;
}

template <typename TN_, typename TA_, typename TH_>
HFSM2_CONSTEXPR(14)
TaskStatus
S_<TN_, TA_, TH_>::deepPostUpdate(FullControl& control) noexcept {
	HFSM2_LOG_STATE_METHOD(&Head::postUpdate,
						   Method::POST_UPDATE);

ScopedOrigin origin{control, STATE_ID};

	Head::	  postUpdate(control);
	Head::widePostUpdate(control);

return control._taskStatus;
}

template <typename TN_, typename TA_, typename TH_>
template <typename TEvent>
HFSM2_CONSTEXPR(14)
TaskStatus
S_<TN_, TA_, TH_>::deepPreReact(EventControl& control,
								const TEvent& event) noexcept
{
auto method = static_cast<void (Head::*)(const TEvent&, EventControl&)>(&Head::preReact);

	HFSM2_LOG_STATE_METHOD(method,
						   Method::PRE_REACT);

ScopedOrigin origin{control, STATE_ID};

	Head::widePreReact(event, control);
(this->*method) (event, control);

return control._taskStatus;
}

template <typename TN_, typename TA_, typename TH_>
template <typename TEvent>
HFSM2_CONSTEXPR(14)
TaskStatus
S_<TN_, TA_, TH_>::deepReact(EventControl& control,
							 const TEvent& event) noexcept
{
auto method = static_cast<void (Head::*)(const TEvent&, EventControl&)>(&Head::react);

	HFSM2_LOG_STATE_METHOD(method,
						   Method::REACT);

ScopedOrigin origin{control, STATE_ID};

	Head::wideReact(event, control);
(this->*method)(event, control);

return control._taskStatus;
}

template <typename TN_, typename TA_, typename TH_>
template <typename TEvent>
HFSM2_CONSTEXPR(14)
TaskStatus
S_<TN_, TA_, TH_>::deepPostReact(EventControl& control,
								 const TEvent& event) noexcept
{
auto method = static_cast<void (Head::*)(const TEvent&, EventControl&)>(&Head::postReact);

	HFSM2_LOG_STATE_METHOD(method,
						   Method::POST_REACT);

ScopedOrigin origin{control, STATE_ID};

(this->*method)	   (event, control);
	Head::widePostReact(event, control);

return control._taskStatus;
}

template <typename TN_, typename TA_, typename TH_>
template <typename TEvent>
HFSM2_CONSTEXPR(14)
void
	S_<TN_, TA_, TH_>::deepQuery(ConstControl& control,
	TEvent&  event) const noexcept
{
	auto method = static_cast<void (Head::*)(TEvent&, ConstControl&) const>(&Head::query);

	HFSM2_LOG_STATE_METHOD(method,
		Method::QUERY);

	ScopedCOrigin origin{control, STATE_ID};

	(this->*method)(event, control);
		Head::wideQuery(event, control);
}

#if HFSM2_PLANS_AVAILABLE()

template <typename TN_, typename TA_, typename TH_>
HFSM2_CONSTEXPR(14)
TaskStatus
S_<TN_, TA_, TH_>::deepUpdatePlans(FullControl& control) noexcept {
	if (control._core.planData.tasksFailures .get(STATE_ID))
		return TaskStatus{TaskStatus::FAILURE};
	else
	if (control._core.planData.tasksSuccesses.get(STATE_ID))
		return TaskStatus{TaskStatus::SUCCESS};
	else
		return TaskStatus{};
}

#endif

template <typename TN_, typename TA_, typename TH_>
HFSM2_CONSTEXPR(14)
bool
S_<TN_, TA_, TH_>::deepExitGuard(GuardControl& control) noexcept {
	HFSM2_LOG_STATE_METHOD(&Head::exitGuard,
						   Method::EXIT_GUARD);

ScopedOrigin origin{control, STATE_ID};

const bool cancelledBefore = control._cancelled;

	Head::wideExitGuard(control);
	Head::	  exitGuard(control);

return !cancelledBefore && control._cancelled;
}

template <typename TN_, typename TA_, typename TH_>
HFSM2_CONSTEXPR(14)
void
S_<TN_, TA_, TH_>::deepExit(PlanControl& control) noexcept {
	HFSM2_LOG_STATE_METHOD(&Head::exit,
						   Method::EXIT);

ScopedOrigin origin{control, STATE_ID};

	// if you see..
	// VS	 - error C2039:  'exit': is not a member of 'Blah'
	// Clang - error : no member named 'exit' in 'Blah'
	//
	// .. inherit state 'Blah' from hfsm2::Machine::Instance::State
	Head::	  exit(control);
	Head::wideExit(control);

	HFSM2_IF_PLANS(control._core.planData.clearTaskStatus(STATE_ID));
}

#if HFSM2_PLANS_AVAILABLE()

template <typename TN_, typename TA_, typename TH_>
HFSM2_CONSTEXPR(14)
void
S_<TN_, TA_, TH_>::wrapPlanSucceeded(FullControl& control) noexcept {
	HFSM2_LOG_STATE_METHOD(&Head::planSucceeded,
						   Method::PLAN_SUCCEEDED);

ScopedOrigin origin{control, STATE_ID};

	Head::planSucceeded(control);
}

template <typename TN_, typename TA_, typename TH_>
HFSM2_CONSTEXPR(14)
void
S_<TN_, TA_, TH_>::wrapPlanFailed(FullControl& control) noexcept {
	HFSM2_LOG_STATE_METHOD(&Head::planFailed,
						   Method::PLAN_FAILED);

ScopedOrigin origin{control, STATE_ID};

	Head::planFailed(control);
}

#endif

template <typename TN_, typename TA_, typename TH_>
HFSM2_CONSTEXPR(14)
void
S_<TN_, TA_, TH_>::deepForwardRequest(Control& HFSM2_IF_TRANSITION_HISTORY(control),
									  const Request HFSM2_IF_TRANSITION_HISTORY(request)) noexcept
{
	HFSM2_IF_TRANSITION_HISTORY(control.pinLastTransition(STATE_ID, request.index));
}

template <typename TN_, typename TA_, typename TH_>
HFSM2_CONSTEXPR(14)
void
S_<TN_, TA_, TH_>::deepRequestChange(Control& HFSM2_IF_TRANSITION_HISTORY(control),
									 const Request HFSM2_IF_TRANSITION_HISTORY(request)) noexcept
{
	HFSM2_IF_TRANSITION_HISTORY(control.pinLastTransition(STATE_ID, request.index));
}

template <typename TN_, typename TA_, typename TH_>
HFSM2_CONSTEXPR(14)
void
S_<TN_, TA_, TH_>::deepRequestRestart(Control& HFSM2_IF_TRANSITION_HISTORY(control),
									  const Request HFSM2_IF_TRANSITION_HISTORY(request)) noexcept
{
	HFSM2_IF_TRANSITION_HISTORY(control.pinLastTransition(STATE_ID, request.index));
}

template <typename TN_, typename TA_, typename TH_>
HFSM2_CONSTEXPR(14)
void
S_<TN_, TA_, TH_>::deepRequestResume(Control& HFSM2_IF_TRANSITION_HISTORY(control),
									 const Request HFSM2_IF_TRANSITION_HISTORY(request)) noexcept
{
	HFSM2_IF_TRANSITION_HISTORY(control.pinLastTransition(STATE_ID, request.index));
}

template <typename TN_, typename TA_, typename TH_>
HFSM2_CONSTEXPR(14)
void
S_<TN_, TA_, TH_>::deepRequestSelect(Control& HFSM2_IF_TRANSITION_HISTORY(control),
									 const Request HFSM2_IF_TRANSITION_HISTORY(request)) noexcept
{
	HFSM2_IF_TRANSITION_HISTORY(control.pinLastTransition(STATE_ID, request.index));
}

#if HFSM2_UTILITY_THEORY_AVAILABLE()

template <typename TN_, typename TA_, typename TH_>
HFSM2_CONSTEXPR(14)
void
S_<TN_, TA_, TH_>::deepRequestUtilize(Control& HFSM2_IF_TRANSITION_HISTORY(control),
									  const Request HFSM2_IF_TRANSITION_HISTORY(request)) noexcept
{
	HFSM2_IF_TRANSITION_HISTORY(control.pinLastTransition(STATE_ID, request.index));
}

template <typename TN_, typename TA_, typename TH_>
HFSM2_CONSTEXPR(14)
void
S_<TN_, TA_, TH_>::deepRequestRandomize(Control& HFSM2_IF_TRANSITION_HISTORY(control),
										const Request HFSM2_IF_TRANSITION_HISTORY(request)) noexcept
{
	HFSM2_IF_TRANSITION_HISTORY(control.pinLastTransition(STATE_ID, request.index));
}

template <typename TN_, typename TA_, typename TH_>
HFSM2_CONSTEXPR(14)
typename S_<TN_, TA_, TH_>::UP
S_<TN_, TA_, TH_>::deepReportChange(Control& control) noexcept {
const Utility utility = wrapUtility(control);

const Parent parent = stateParent(control);

return {utility, parent.prong};
}

template <typename TN_, typename TA_, typename TH_>
HFSM2_CONSTEXPR(14)
typename S_<TN_, TA_, TH_>::UP
S_<TN_, TA_, TH_>::deepReportUtilize(Control& control) noexcept {
const Utility utility = wrapUtility(control);
const Parent  parent  = stateParent(control);

return {utility, parent.prong};
}

template <typename TN_, typename TA_, typename TH_>
HFSM2_CONSTEXPR(14)
typename S_<TN_, TA_, TH_>::Rank
S_<TN_, TA_, TH_>::deepReportRank(Control& control) noexcept {
	return wrapRank(control);
}

template <typename TN_, typename TA_, typename TH_>
HFSM2_CONSTEXPR(14)
typename S_<TN_, TA_, TH_>::Utility
S_<TN_, TA_, TH_>::deepReportRandomize(Control& control) noexcept {
	return wrapUtility(control);
}

#endif

#if HFSM2_STRUCTURE_REPORT_AVAILABLE()

template <typename TN_, typename TA_, typename TH_>
HFSM2_CONSTEXPR(NO)
const char*
S_<TN_, TA_, TH_>::name() noexcept {
const std::type_index type = typeid(Head);
const char* const raw = type.name();

#if defined(_MSC_VER)

	Short first =
		raw[0] == 's' ? 7 : // Struct
		raw[0] == 'c' ? 6 : // Class
						0;

for (Short c = first; raw[c]; ++c)
if (raw[c] == ':')
first = c + 1;

return raw + first;

#elif defined(__clang__) || defined(__GNUC__) || defined(__GNUG__)

return raw;

#else

return raw;

#endif
}

template <typename TN_, typename TA_, typename TH_>
HFSM2_CONSTEXPR(14)
void
	S_<TN_, TA_, TH_>::deepGetNames(const Long parent,
	const RegionType region,
	const Short depth,
	StructureStateInfos& stateInfos) const noexcept
{
	stateInfos.emplace(StructureStateInfo{parent, region, depth, name()});
		}

#endif

}
}

namespace hfsm2 {
	namespace detail {

#if HFSM2_DEBUG_STATE_TYPE_AVAILABLE() || HFSM2_STRUCTURE_REPORT_AVAILABLE() || HFSM2_LOG_INTERFACE_AVAILABLE()

		struct None final {};

#endif

	template <
	typename TIndices
	, typename TArgs
	>
	struct S_<TIndices, TArgs, EmptyT<TArgs>>
		: EmptyT<TArgs>
		{
		static constexpr StateID STATE_ID = TIndices::STATE_ID;

		using Context		= typename TArgs::Context;

#if HFSM2_UTILITY_THEORY_AVAILABLE()
		using Rank			= typename TArgs::Rank;
		using Utility		= typename TArgs::Utility;
		using UP			= typename TArgs::UP;
#endif

#if HFSM2_LOG_INTERFACE_AVAILABLE()
		using Logger		= typename TArgs::Logger;
#endif

		using ConstControl	= ConstControlT<TArgs>;
		using ScopedCOrigin	= typename ConstControl::Origin;

		using Control		= ControlT	   <TArgs>;
		using Registry		= RegistryT	   <TArgs>;
		using StateParents	= typename Registry::StateParents;

		using PlanControl	= PlanControlT <TArgs>;
		using ScopedOrigin	= typename PlanControl::Origin;

		using FullControl	= FullControlT <TArgs>;
		using GuardControl	= GuardControlT<TArgs>;
		using EventControl	= EventControlT<TArgs>;

		using Empty			= EmptyT<TArgs>;
		using Head			= Empty;

	HFSM2_CONSTEXPR(14)	Parent		 stateParent		  (		Control& control)								noexcept	{ return control._core.registry.stateParents[STATE_ID];	}

	HFSM2_CONSTEXPR(14)	void		 deepRegister		  (	   Registry& registry, const Parent parent)			noexcept;

	HFSM2_CONSTEXPR(14)	Prong		 wrapSelect			  (		Control& control)								noexcept;

#if HFSM2_UTILITY_THEORY_AVAILABLE()
	HFSM2_CONSTEXPR(14)	Rank		 wrapRank			  (		Control& control)								noexcept;
	HFSM2_CONSTEXPR(14)	Utility		 wrapUtility		  (		Control& control)								noexcept;
#endif

HFSM2_CONSTEXPR(14)	bool		 deepForwardEntryGuard(GuardControl&		)								noexcept	{ return false;		}
	HFSM2_CONSTEXPR(14)	bool		 deepEntryGuard		  (GuardControl& control)								noexcept;

	HFSM2_CONSTEXPR(14)	void		 deepEnter			  ( PlanControl& control)								noexcept;
	HFSM2_CONSTEXPR(14)	void		 deepReenter		  ( PlanControl& control)								noexcept;

	HFSM2_CONSTEXPR(14)	TaskStatus	 deepPreUpdate		  ( FullControl& control)								noexcept;
	HFSM2_CONSTEXPR(14)	TaskStatus	 deepUpdate			  ( FullControl& control)								noexcept;
	HFSM2_CONSTEXPR(14)	TaskStatus	 deepPostUpdate		  ( FullControl& control)								noexcept;

	template <typename TEvent>
	HFSM2_CONSTEXPR(14)	TaskStatus	 deepPreReact		  (EventControl& control, const TEvent&	event)			noexcept;

	template <typename TEvent>
	HFSM2_CONSTEXPR(14)	TaskStatus	 deepReact			  (EventControl& control, const TEvent&	event)			noexcept;

	template <typename TEvent>
	HFSM2_CONSTEXPR(14)	TaskStatus	 deepPostReact		  (EventControl& control, const TEvent&	event)			noexcept;

	template <typename TEvent>
	HFSM2_CONSTEXPR(14)	void		 deepQuery			  (ConstControl& control,		TEvent& event)	  const noexcept;

#if HFSM2_PLANS_AVAILABLE()
	HFSM2_CONSTEXPR(14)	TaskStatus	 deepUpdatePlans	  ( FullControl& control)								noexcept;
#endif

	HFSM2_CONSTEXPR(14)	bool		 deepForwardExitGuard (GuardControl&		)								noexcept	{ return false;		}
	HFSM2_CONSTEXPR(14)	bool		 deepExitGuard		  (GuardControl& control)								noexcept;

	HFSM2_CONSTEXPR(14)	void		 deepExit			  ( PlanControl& control)								noexcept;

#if HFSM2_PLANS_AVAILABLE()
	HFSM2_CONSTEXPR(14)	void		 wrapPlanSucceeded	  ( FullControl& control)								noexcept;
	HFSM2_CONSTEXPR(14)	void		 wrapPlanFailed		  ( FullControl& control)								noexcept;
#endif

	HFSM2_CONSTEXPR(14)	void		 deepForwardActive	  (	   Control&,		 const Request		  )			noexcept	{}
	HFSM2_CONSTEXPR(14)	void		 deepForwardRequest	  (	   Control& control, const Request request)			noexcept;

	HFSM2_CONSTEXPR(14)	void		 deepRequestChange	  (	    Control& control, const Request request)		noexcept;
	HFSM2_CONSTEXPR(14)	void		 deepRequestRestart	  (		Control& control, const Request request)		noexcept;
	HFSM2_CONSTEXPR(14)	void		 deepRequestResume	  (		Control& control, const Request request)		noexcept;
	HFSM2_CONSTEXPR(14)	void		 deepRequestSelect	  (	    Control& control, const Request request)		noexcept;

#if HFSM2_UTILITY_THEORY_AVAILABLE()
	HFSM2_CONSTEXPR(14)	void		 deepRequestUtilize	  (		Control& control, const Request request)		noexcept;
	HFSM2_CONSTEXPR(14)	void		 deepRequestRandomize (		Control& control, const Request request)		noexcept;

	HFSM2_CONSTEXPR(14)	UP			 deepReportChange	  (	    Control& control)								noexcept;
	HFSM2_CONSTEXPR(14)	UP			 deepReportUtilize	  (	    Control& control)								noexcept;
	HFSM2_CONSTEXPR(14)	Rank		 deepReportRank		  (		Control& control)								noexcept;
	HFSM2_CONSTEXPR(14)	Utility		 deepReportRandomize  (	    Control& control)								noexcept;
#endif

	HFSM2_CONSTEXPR(14)	void		 deepChangeToRequested(	    Control&		)								noexcept	{}

#if HFSM2_SERIALIZATION_AVAILABLE()
	using WriteStream	= typename TArgs::WriteStream;
	using ReadStream	= typename TArgs::ReadStream;

	HFSM2_CONSTEXPR(14)	void		 deepSaveActive		  (const Registry&, WriteStream&)				  const noexcept	{}
	HFSM2_CONSTEXPR(14)	void		 deepSaveResumable	  (const Registry&, WriteStream&)				  const noexcept	{}

	HFSM2_CONSTEXPR(14)	void		 deepLoadRequested	  (		 Registry&,  ReadStream&)				  const noexcept	{}
	HFSM2_CONSTEXPR(14)	void		 deepLoadResumable	  (		 Registry&,  ReadStream&)				  const noexcept	{}
#endif

#if HFSM2_STRUCTURE_REPORT_AVAILABLE()
	using StructureStateInfos = typename TArgs::StructureStateInfos;

	static
	HFSM2_CONSTEXPR(NO)	const char* name() noexcept;

	HFSM2_CONSTEXPR(14)	void deepGetNames(const Long parent,
										  const RegionType region,
										  const Short depth,
										  StructureStateInfos& stateInfos)							  const noexcept;
#endif

#if HFSM2_DEBUG_STATE_TYPE_AVAILABLE() || HFSM2_STRUCTURE_REPORT_AVAILABLE() || HFSM2_LOG_INTERFACE_AVAILABLE()

	HFSM2_IF_TYPEINDEX(const std::type_index TYPE = typeid(None));

static constexpr Long NAME_COUNT = 0;

#endif

#if HFSM2_LOG_INTERFACE_AVAILABLE()

	template <typename TReturn, typename... TParams>
	HFSM2_CONSTEXPR(14)
	void log(TReturn (Empty::*)(TParams...),
			 Logger&,
			 const Context&,
			 const Method)																			  const noexcept
	{}

	template <typename TReturn, typename... TParams>
	HFSM2_CONSTEXPR(14)
	void log(TReturn (Empty::*)(TParams...) const,
Logger&,
const Context&,
			 const Method)																			  const noexcept
	{}

#endif
};

}
}

namespace hfsm2 {
	namespace detail {

		template <typename TN_, typename TA_>
		HFSM2_CONSTEXPR(14)
		void
		S_<TN_, TA_, EmptyT<TA_>>::deepRegister(Registry& registry,
		const Parent parent) noexcept
		{
		registry.stateParents[STATE_ID] = parent;
	}

	template <typename TN_, typename TA_>
	HFSM2_CONSTEXPR(14)
	Prong
	S_<TN_, TA_, EmptyT<TA_>>::wrapSelect(Control& HFSM2_IF_LOG_STATE_METHOD(control)) noexcept {
	HFSM2_LOG_STATE_METHOD(&Empty::select,
	Method::SELECT);

	return INVALID_PRONG;
}

#if HFSM2_UTILITY_THEORY_AVAILABLE()

template <typename TN_, typename TA_>
HFSM2_CONSTEXPR(14)
typename S_<TN_, TA_, EmptyT<TA_>>::Rank
S_<TN_, TA_, EmptyT<TA_>>::wrapRank(Control& HFSM2_IF_LOG_STATE_METHOD(control)) noexcept {
	HFSM2_LOG_STATE_METHOD(&Empty::rank,
						   Method::RANK);

	return Rank{};
}

template <typename TN_, typename TA_>
HFSM2_CONSTEXPR(14)
typename S_<TN_, TA_, EmptyT<TA_>>::Utility
S_<TN_, TA_, EmptyT<TA_>>::wrapUtility(Control& HFSM2_IF_LOG_STATE_METHOD(control)) noexcept {
	HFSM2_LOG_STATE_METHOD(&Empty::utility,
						   Method::UTILITY);

	return Utility{};
}

#endif

template <typename TN_, typename TA_>
HFSM2_CONSTEXPR(14)
bool
S_<TN_, TA_, EmptyT<TA_>>::deepEntryGuard(GuardControl& HFSM2_IF_LOG_STATE_METHOD(control)) noexcept {
	HFSM2_LOG_STATE_METHOD(&Empty::entryGuard,
						   Method::ENTRY_GUARD);

	return false;
}

template <typename TN_, typename TA_>
HFSM2_CONSTEXPR(14)
void
S_<TN_, TA_, EmptyT<TA_>>::deepEnter(PlanControl& HFSM2_IF_LOG_STATE_METHOD(control)) noexcept {
	HFSM2_LOG_STATE_METHOD(&Empty::enter,
						   Method::ENTER);
}

template <typename TN_, typename TA_>
HFSM2_CONSTEXPR(14)
void
S_<TN_, TA_, EmptyT<TA_>>::deepReenter(PlanControl& HFSM2_IF_LOG_STATE_METHOD(control)) noexcept {
	HFSM2_LOG_STATE_METHOD(&Empty::reenter,
						   Method::REENTER);
}

template <typename TN_, typename TA_>
HFSM2_CONSTEXPR(14)
TaskStatus
S_<TN_, TA_, EmptyT<TA_>>::deepPreUpdate(FullControl& HFSM2_IF_LOG_STATE_METHOD(control)) noexcept {
	HFSM2_LOG_STATE_METHOD(&Empty::preUpdate,
						   Method::PRE_UPDATE);

	return TaskStatus{};
}

template <typename TN_, typename TA_>
HFSM2_CONSTEXPR(14)
TaskStatus
S_<TN_, TA_, EmptyT<TA_>>::deepUpdate(FullControl& HFSM2_IF_LOG_STATE_METHOD(control)) noexcept {
	HFSM2_LOG_STATE_METHOD(&Empty::update,
						   Method::UPDATE);

	return TaskStatus{};
}

template <typename TN_, typename TA_>
HFSM2_CONSTEXPR(14)
TaskStatus
S_<TN_, TA_, EmptyT<TA_>>::deepPostUpdate(FullControl& HFSM2_IF_LOG_STATE_METHOD(control)) noexcept {
	HFSM2_LOG_STATE_METHOD(&Empty::postUpdate,
						   Method::POST_UPDATE);

	return TaskStatus{};
}

template <typename TN_, typename TA_>
template <typename TEvent>
HFSM2_CONSTEXPR(14)
TaskStatus
S_<TN_, TA_, EmptyT<TA_>>::deepPreReact(EventControl& HFSM2_IF_LOG_STATE_METHOD(control),
										const TEvent& HFSM2_UNUSED(event)) noexcept
{
	HFSM2_LOG_STATE_METHOD(static_cast<void (Empty::*)(const TEvent&, EventControl&)>(&Empty::preReact),
						   Method::PRE_REACT);

	return TaskStatus{};
}

template <typename TN_, typename TA_>
template <typename TEvent>
HFSM2_CONSTEXPR(14)
TaskStatus
S_<TN_, TA_, EmptyT<TA_>>::deepReact(EventControl& HFSM2_IF_LOG_STATE_METHOD(control),
									 const TEvent& HFSM2_UNUSED(event)) noexcept
{
	HFSM2_LOG_STATE_METHOD(static_cast<void (Empty::*)(const TEvent&, EventControl&)>(&Empty::react),
						   Method::REACT);

	return TaskStatus{};
}

template <typename TN_, typename TA_>
template <typename TEvent>
HFSM2_CONSTEXPR(14)
TaskStatus
S_<TN_, TA_, EmptyT<TA_>>::deepPostReact(EventControl& HFSM2_IF_LOG_STATE_METHOD(control),
										 const TEvent& HFSM2_UNUSED(event)) noexcept
{
	HFSM2_LOG_STATE_METHOD(static_cast<void (Empty::*)(const TEvent&, EventControl&)>(&Empty::postReact),
						   Method::POST_REACT);

	return TaskStatus{};
}

template <typename TN_, typename TA_>
template <typename TEvent>
HFSM2_CONSTEXPR(14)
void
S_<TN_, TA_, EmptyT<TA_>>::deepQuery(ConstControl& HFSM2_IF_LOG_STATE_METHOD(control),
									 TEvent& HFSM2_UNUSED(event)) const noexcept
{
	HFSM2_LOG_STATE_METHOD(static_cast<void (Empty::*)(TEvent&, ConstControl&) const>(&Empty::query),
						   Method::QUERY);
}

#if HFSM2_PLANS_AVAILABLE()

template <typename TN_, typename TA_>
HFSM2_CONSTEXPR(14)
TaskStatus
S_<TN_, TA_, EmptyT<TA_>>::deepUpdatePlans(FullControl& control) noexcept {
	if (control._core.planData.tasksFailures .get(STATE_ID))
		return TaskStatus{TaskStatus::FAILURE};
	else
	if (control._core.planData.tasksSuccesses.get(STATE_ID))
		return TaskStatus{TaskStatus::SUCCESS};
	else
		return TaskStatus{};
}

#endif

template <typename TN_, typename TA_>
HFSM2_CONSTEXPR(14)
bool
S_<TN_, TA_, EmptyT<TA_>>::deepExitGuard(GuardControl& HFSM2_IF_LOG_STATE_METHOD(control)) noexcept {
	HFSM2_LOG_STATE_METHOD(&Empty::exitGuard,
						   Method::EXIT_GUARD);

	return false;
}

template <typename TN_, typename TA_>
HFSM2_CONSTEXPR(14)
void
S_<TN_, TA_, EmptyT<TA_>>::deepExit(PlanControl& HFSM2_IF_LOG_STATE_METHOD(control)) noexcept {
	HFSM2_LOG_STATE_METHOD(&Empty::exit,
						   Method::EXIT);
}

#if HFSM2_PLANS_AVAILABLE()

template <typename TN_, typename TA_>
HFSM2_CONSTEXPR(14)
void
S_<TN_, TA_, EmptyT<TA_>>::wrapPlanSucceeded(FullControl& HFSM2_IF_LOG_STATE_METHOD(control)) noexcept {
	HFSM2_LOG_STATE_METHOD(&Empty::planSucceeded,
						   Method::PLAN_SUCCEEDED);
}

template <typename TN_, typename TA_>
HFSM2_CONSTEXPR(14)
void
S_<TN_, TA_, EmptyT<TA_>>::wrapPlanFailed(FullControl& HFSM2_IF_LOG_STATE_METHOD(control)) noexcept {
	HFSM2_LOG_STATE_METHOD(&Empty::planFailed,
						   Method::PLAN_FAILED);
}

#endif

template <typename TN_, typename TA_>
HFSM2_CONSTEXPR(14)
void
S_<TN_, TA_, EmptyT<TA_>>::deepForwardRequest(Control& HFSM2_IF_TRANSITION_HISTORY(control),
											  const Request HFSM2_IF_TRANSITION_HISTORY(request)) noexcept
{
	HFSM2_IF_TRANSITION_HISTORY(control.pinLastTransition(STATE_ID, request.index));
}

template <typename TN_, typename TA_>
HFSM2_CONSTEXPR(14)
void
S_<TN_, TA_, EmptyT<TA_>>::deepRequestChange(Control& HFSM2_IF_TRANSITION_HISTORY(control),
											 const Request HFSM2_IF_TRANSITION_HISTORY(request)) noexcept
{
	HFSM2_IF_TRANSITION_HISTORY(control.pinLastTransition(STATE_ID, request.index));
}

template <typename TN_, typename TA_>
HFSM2_CONSTEXPR(14)
void
S_<TN_, TA_, EmptyT<TA_>>::deepRequestRestart(Control& HFSM2_IF_TRANSITION_HISTORY(control),
											  const Request HFSM2_IF_TRANSITION_HISTORY(request)) noexcept
{
	HFSM2_IF_TRANSITION_HISTORY(control.pinLastTransition(STATE_ID, request.index));
}

template <typename TN_, typename TA_>
HFSM2_CONSTEXPR(14)
void
S_<TN_, TA_, EmptyT<TA_>>::deepRequestResume(Control& HFSM2_IF_TRANSITION_HISTORY(control),
											 const Request HFSM2_IF_TRANSITION_HISTORY(request)) noexcept
{
	HFSM2_IF_TRANSITION_HISTORY(control.pinLastTransition(STATE_ID, request.index));
}

template <typename TN_, typename TA_>
HFSM2_CONSTEXPR(14)
void
S_<TN_, TA_, EmptyT<TA_>>::deepRequestSelect(Control& HFSM2_IF_TRANSITION_HISTORY(control),
											 const Request HFSM2_IF_TRANSITION_HISTORY(request)) noexcept
{
	HFSM2_IF_TRANSITION_HISTORY(control.pinLastTransition(STATE_ID, request.index));
}

#if HFSM2_UTILITY_THEORY_AVAILABLE()

template <typename TN_, typename TA_>
HFSM2_CONSTEXPR(14)
void
S_<TN_, TA_, EmptyT<TA_>>::deepRequestUtilize(Control& HFSM2_IF_TRANSITION_HISTORY(control),
											  const Request HFSM2_IF_TRANSITION_HISTORY(request)) noexcept
{
	HFSM2_IF_TRANSITION_HISTORY(control.pinLastTransition(STATE_ID, request.index));
}

template <typename TN_, typename TA_>
HFSM2_CONSTEXPR(14)
void
S_<TN_, TA_, EmptyT<TA_>>::deepRequestRandomize(Control& HFSM2_IF_TRANSITION_HISTORY(control),
												const Request HFSM2_IF_TRANSITION_HISTORY(request)) noexcept
{
	HFSM2_IF_TRANSITION_HISTORY(control.pinLastTransition(STATE_ID, request.index));
}

template <typename TN_, typename TA_>
HFSM2_CONSTEXPR(14)
typename S_<TN_, TA_, EmptyT<TA_>>::UP
S_<TN_, TA_, EmptyT<TA_>>::deepReportChange(Control& control) noexcept {
const Parent parent = stateParent(control);

	return {Utility{}, parent.prong};
}

template <typename TN_, typename TA_>
HFSM2_CONSTEXPR(14)
typename S_<TN_, TA_, EmptyT<TA_>>::UP
S_<TN_, TA_, EmptyT<TA_>>::deepReportUtilize(Control& control) noexcept {
const Parent parent  = stateParent(control);

	return {Utility{}, parent.prong};
}

template <typename TN_, typename TA_>
HFSM2_CONSTEXPR(14)
typename S_<TN_, TA_, EmptyT<TA_>>::Rank
S_<TN_, TA_, EmptyT<TA_>>::deepReportRank(Control& HFSM2_UNUSED(control)) noexcept {
	return Rank{};
}

template <typename TN_, typename TA_>
HFSM2_CONSTEXPR(14)
typename S_<TN_, TA_, EmptyT<TA_>>::Utility
S_<TN_, TA_, EmptyT<TA_>>::deepReportRandomize(Control& HFSM2_UNUSED(control)) noexcept {
	return Utility{};
}

#endif

#if HFSM2_STRUCTURE_REPORT_AVAILABLE()

template <typename TN_, typename TA_>
HFSM2_CONSTEXPR(NO)
const char*
S_<TN_, TA_, EmptyT<TA_>>::name() noexcept {
	return "";
}

template <typename TN_, typename TA_>
HFSM2_CONSTEXPR(14)
void
	S_<TN_, TA_, EmptyT<TA_>>::deepGetNames(const Long parent,
	const RegionType region,
	const Short depth,
	StructureStateInfos& stateInfos) const noexcept
{
	stateInfos.emplace(StructureStateInfo{parent, region, depth, name()});
		}

#endif

}
}

namespace hfsm2 {
	namespace detail {

		template <typename>
		struct SI_;

		template <Strategy, typename, typename...>
		struct CI_;

		template <typename>
		struct CSI_;

		template <typename, typename...>
		struct OI_;

		template <typename...>
		struct OSI_;

		template <typename TI, typename... TR>
		struct OSI_<TI, TR...>;

		template <typename TI>
		struct OSI_<TI>;

		template <typename...>
		struct WrapInfoT;

		template <typename TH>
		struct WrapInfoT	<TH> final {
			using Type = SI_<TH>;
		};

		template <Strategy SG, typename TH, typename... TS>
		struct WrapInfoT<CI_<SG, TH, TS...>> final {
			using Type = CI_<SG, TH, TS...>;
		};

		template <typename... TS>
		struct WrapInfoT<OI_<TS...>> final {
			using Type = OI_<TS...>;
		};

		template <typename... TS>
		using WrapInfo = typename WrapInfoT<TS...>::Type;

		template <typename THead>
		struct SI_ final {
			using Head				= THead;
			using StateList			= TL_<Head>;
			using RegionList		= TL_<>;

			static constexpr Short WIDTH		  = 1;
			static constexpr Long  REVERSE_DEPTH  = 1;
			static constexpr Short COMPO_COUNT	  = 0;
			static constexpr Long  COMPO_PRONGS	  = 0;
			static constexpr Short ORTHO_COUNT	  = 0;
			static constexpr Short ORTHO_UNITS	  = 0;

			static constexpr Long  STATE_COUNT	  =  StateList::SIZE;
			static constexpr Short REGION_COUNT	  = RegionList::SIZE;

#if HFSM2_SERIALIZATION_AVAILABLE()
			static constexpr Long  ACTIVE_BITS	  = 0;
			static constexpr Long  RESUMABLE_BITS = 0;
#endif
		};

		template <Strategy TStrategy, typename THead, typename... TSubStates>
		struct CI_ final {
		static constexpr Strategy STRATEGY = TStrategy;

		using Head				= THead;
		using HeadInfo			= SI_<Head>;
		using SubStates			= CSI_<TL_<TSubStates...>>;
		using StateList			= Merge<typename HeadInfo::StateList, typename SubStates::StateList>;
		using RegionList		= Merge<typename HeadInfo::StateList, typename SubStates::RegionList>;

		static constexpr Short WIDTH		  = sizeof...(TSubStates);
		static constexpr Long  REVERSE_DEPTH  = SubStates::REVERSE_DEPTH + 1;
		static constexpr Short COMPO_COUNT	  = SubStates::COMPO_COUNT	 + 1;
		static constexpr Long  COMPO_PRONGS	  = SubStates::COMPO_PRONGS	 + WIDTH;
		static constexpr Short ORTHO_COUNT	  = SubStates::ORTHO_COUNT;
		static constexpr Short ORTHO_UNITS	  = SubStates::ORTHO_UNITS;

		static constexpr Long  STATE_COUNT	  =  StateList::SIZE;
		static constexpr Short REGION_COUNT	  = RegionList::SIZE;

#if HFSM2_SERIALIZATION_AVAILABLE()
		static constexpr Long  WIDTH_BITS	  = bitContain(WIDTH);
		static constexpr Long  ACTIVE_BITS	  = SubStates::ACTIVE_BITS	  + WIDTH_BITS;
		static constexpr Long  RESUMABLE_BITS = SubStates::RESUMABLE_BITS + WIDTH_BITS + 1;
#endif
	};

	template <typename TI, typename... TR>
	struct CSI_<TL_<TI, TR...>> final {
		using Initial			= WrapInfo<TI>;
		using Remaining			= CSI_<TL_<TR...>>;
		using StateList			= Merge<typename Initial::StateList,  typename Remaining::StateList>;
		using RegionList		= Merge<typename Initial::RegionList, typename Remaining::RegionList>;

		static constexpr Long  REVERSE_DEPTH  = max(Initial::REVERSE_DEPTH,	  Remaining::REVERSE_DEPTH);
		static constexpr Short COMPO_COUNT	  =		Initial::COMPO_COUNT	+ Remaining::COMPO_COUNT;
		static constexpr Long  COMPO_PRONGS	  =		Initial::COMPO_PRONGS	+ Remaining::COMPO_PRONGS;
		static constexpr Short ORTHO_COUNT	  =		Initial::ORTHO_COUNT	+ Remaining::ORTHO_COUNT;
		static constexpr Short ORTHO_UNITS	  =		Initial::ORTHO_UNITS	+ Remaining::ORTHO_UNITS;

		static constexpr Long  STATE_COUNT	  =  StateList::SIZE;
		static constexpr Short REGION_COUNT	  = RegionList::SIZE;

#if HFSM2_SERIALIZATION_AVAILABLE()
		static constexpr Long  ACTIVE_BITS	  = max(Initial::ACTIVE_BITS,	  Remaining::ACTIVE_BITS);
		static constexpr Long  RESUMABLE_BITS =		Initial::RESUMABLE_BITS + Remaining::RESUMABLE_BITS;
#endif
	};

	template <typename TI>
	struct CSI_<TL_<TI>> final {
		using Initial			= WrapInfo<TI>;
		using StateList			= typename Initial::StateList;
		using RegionList		= typename Initial::RegionList;

		static constexpr Long  REVERSE_DEPTH  = Initial::REVERSE_DEPTH;
		static constexpr Short COMPO_COUNT	  = Initial::COMPO_COUNT;
		static constexpr Long  COMPO_PRONGS	  = Initial::COMPO_PRONGS;
		static constexpr Short ORTHO_COUNT	  = Initial::ORTHO_COUNT;
		static constexpr Short ORTHO_UNITS	  = Initial::ORTHO_UNITS;

		static constexpr Long  STATE_COUNT	  =  StateList::SIZE;
		static constexpr Short REGION_COUNT	  = RegionList::SIZE;

#if HFSM2_SERIALIZATION_AVAILABLE()
		static constexpr Long  ACTIVE_BITS	  = Initial::ACTIVE_BITS;
		static constexpr Long  RESUMABLE_BITS = Initial::RESUMABLE_BITS;
#endif
	};

	template <typename THead, typename... TSubStates>
	struct OI_ final {
	using Head				= THead;
	using HeadInfo			= SI_<Head>;
	using SubStates			= OSI_<TSubStates...>;
	using StateList			= Merge<typename HeadInfo::StateList, typename SubStates::StateList>;
	using RegionList		= Merge<typename HeadInfo::StateList, typename SubStates::RegionList>;

	static constexpr Short WIDTH			= sizeof...(TSubStates);
	static constexpr Long  REVERSE_DEPTH	= SubStates::REVERSE_DEPTH + 1;
	static constexpr Short COMPO_COUNT		= SubStates::COMPO_COUNT;
	static constexpr Long  COMPO_PRONGS		= SubStates::COMPO_PRONGS;
	static constexpr Short ORTHO_COUNT		= SubStates::ORTHO_COUNT   + 1;
	static constexpr Short ORTHO_UNITS		= SubStates::ORTHO_UNITS   + contain(WIDTH, 8);

	static constexpr Long  STATE_COUNT		=  StateList::SIZE;
	static constexpr Short REGION_COUNT		= RegionList::SIZE;

#if HFSM2_SERIALIZATION_AVAILABLE()
	static constexpr Long  ACTIVE_BITS		= SubStates::ACTIVE_BITS;
	static constexpr Long  RESUMABLE_BITS	= SubStates::RESUMABLE_BITS;
#endif
};

template <typename TI, typename... TR>
struct OSI_<TI, TR...> final {
	using Initial			= WrapInfo<TI>;
	using Remaining			= OSI_<TR...>;
	using StateList			= Merge<typename Initial::StateList,  typename Remaining::StateList>;
	using RegionList		= Merge<typename Initial::RegionList, typename Remaining::RegionList>;

	static constexpr Long  REVERSE_DEPTH  = max(Initial::REVERSE_DEPTH,	  Remaining::REVERSE_DEPTH);
	static constexpr Short COMPO_COUNT	  =		Initial::COMPO_COUNT	+ Remaining::COMPO_COUNT;
	static constexpr Long  COMPO_PRONGS	  =		Initial::COMPO_PRONGS	+ Remaining::COMPO_PRONGS;
	static constexpr Short ORTHO_COUNT	  =		Initial::ORTHO_COUNT	+ Remaining::ORTHO_COUNT;
	static constexpr Short ORTHO_UNITS	  =		Initial::ORTHO_UNITS	+ Remaining::ORTHO_UNITS;

#if HFSM2_SERIALIZATION_AVAILABLE()
	static constexpr Long  ACTIVE_BITS	  =		Initial::ACTIVE_BITS    + Remaining::ACTIVE_BITS;
	static constexpr Long  RESUMABLE_BITS =		Initial::RESUMABLE_BITS + Remaining::RESUMABLE_BITS;
#endif
};

template <typename TI>
struct OSI_<TI> final {
	using Initial			= WrapInfo<TI>;
	using StateList			= typename Initial::StateList;
	using RegionList		= typename Initial::RegionList;

	static constexpr Long  REVERSE_DEPTH	= Initial::REVERSE_DEPTH;
	static constexpr Short COMPO_COUNT		= Initial::COMPO_COUNT;
	static constexpr Long  COMPO_PRONGS		= Initial::COMPO_PRONGS;
	static constexpr Short ORTHO_COUNT		= Initial::ORTHO_COUNT;
	static constexpr Short ORTHO_UNITS		= Initial::ORTHO_UNITS;

#if HFSM2_SERIALIZATION_AVAILABLE()
	static constexpr Long  ACTIVE_BITS		= Initial::ACTIVE_BITS;
	static constexpr Long  RESUMABLE_BITS	= Initial::RESUMABLE_BITS;
#endif
};

template <
	typename TConfig
  , typename TStateList
  , typename TRegionList
  , Long NCompoCount
  , Long NOrthoCount
  , Long NOrthoUnits
  , typename TReactOrder
  HFSM2_IF_SERIALIZATION(, Long NSerialBits)
  HFSM2_IF_PLANS(, Long NTaskCapacity)
  , typename TPayload
>
struct ArgsT final {
	using Config		= TConfig;
using Context		= typename Config::Context;
	using PureContext	= Undecorate<Context>;

#if HFSM2_UTILITY_THEORY_AVAILABLE()
	using Rank			= typename Config::Rank;
	using Utility		= typename Config::Utility;
	using RNG			= typename Config::RNG;
	using UP			= typename Config::UP;
#endif

#if HFSM2_LOG_INTERFACE_AVAILABLE()
	using Logger		= typename Config::LoggerInterface;
#endif

	using StateList		= TStateList;
using RegionList	= TRegionList;

static constexpr Long  STATE_COUNT			= StateList ::SIZE;
static constexpr Short REGION_COUNT			= RegionList::SIZE;

static constexpr Short COMPO_COUNT			= NCompoCount;
static constexpr Short ORTHO_COUNT			= NOrthoCount;
static constexpr Short ORTHO_UNITS			= NOrthoUnits;

	using ReactOrder	= TReactOrder;

#if HFSM2_SERIALIZATION_AVAILABLE()
	static constexpr Short SERIAL_BITS			= NSerialBits;
#endif

static constexpr Short SUBSTITUTION_LIMIT	= Config::SUBSTITUTION_LIMIT;

#if HFSM2_PLANS_AVAILABLE()
static constexpr Long  TASK_CAPACITY		= NTaskCapacity;
#endif

	using Payload		= TPayload;

#if HFSM2_SERIALIZATION_AVAILABLE()
	using SerialBuffer	= StreamBufferT  <SERIAL_BITS>;
	using WriteStream	= BitWriteStreamT<SERIAL_BITS>;
	using ReadStream	= BitReadStreamT <SERIAL_BITS>;
#endif

	HFSM2_IF_STRUCTURE_REPORT(using StructureStateInfos = DynamicArrayT<StructureStateInfo, STATE_COUNT>);
};

template <StateID NStateID,
		  Short NCompoIndex,
		  Short NOrthoIndex,
		  Short NOrthoUnit>
struct I_ final {
	static constexpr StateID STATE_ID	 = NStateID;
	static constexpr Short	 COMPO_INDEX = NCompoIndex;
	static constexpr Short	 ORTHO_INDEX = NOrthoIndex;
	static constexpr Short	 ORTHO_UNIT	 = NOrthoUnit;
};

template <typename, typename, typename>
struct S_;

template <typename, typename, Strategy, typename, typename...>
struct C_;

template <typename, typename, Strategy, Prong, typename>
struct CS_;

template <typename, typename, typename, typename...>
struct O_;

template <typename, typename, Prong, typename...>
struct OS_;

template <typename, typename>
class InstanceT;

template <typename, typename...>
struct MaterialT_;

template <typename TN, typename TA, typename TH>
struct MaterialT_  <TN, TA, TH> final {
	using Type = S_<TN, TA, TH>;
};

template <typename TN, typename TA, Strategy SG, 			  typename... TS>
struct MaterialT_  <TN, TA, CI_<SG, void	  , TS...>> final {
	using Type = C_<TN, TA,     SG, EmptyT<TA>, TS...>;
};

template <typename TN, typename TA, Strategy SG, typename TH, typename... TS>
struct MaterialT_  <TN, TA, CI_<SG, TH,	TS...>> final {
	using Type = C_<TN, TA,     SG, TH,	TS...>;
};

template <typename TN, typename TA,				 typename... TS>
struct MaterialT_  <TN, TA, OI_<void,       TS...>> final {
	using Type = O_<TN, TA,     EmptyT<TA>, TS...>;
};

template <typename TN, typename TA, typename TH, typename... TS>
struct MaterialT_  <TN, TA, OI_<TH, TS...>> final {
	using Type = O_<TN, TA,     TH, TS...>;
};

template <typename TN, typename... TS>
using MaterialT = typename MaterialT_<TN, TS...>::Type;

template <
	typename TConfig
  , typename TApex
>
struct RF_ final {
	using Config			= TConfig;
	using Context			= typename Config::Context;
	using Apex				= TApex;

	using ReactOrder		= typename Config::ReactOrder;

	using StateList			= typename Apex::StateList;
	using RegionList		= typename Apex::RegionList;

	static constexpr Long  STATE_COUNT			= Apex::STATE_COUNT;
	static constexpr Short REGION_COUNT			= Apex::REGION_COUNT;

	static constexpr Short SUBSTITUTION_LIMIT	= Config::SUBSTITUTION_LIMIT;

#if HFSM2_PLANS_AVAILABLE()
	static constexpr Long  TASK_CAPACITY		= Config::TASK_CAPACITY != INVALID_LONG ?
		Config::TASK_CAPACITY : Apex::COMPO_PRONGS * 2;
#endif

	using Payload			= typename Config::Payload;

	static constexpr Short COMPO_COUNT			= Apex::COMPO_COUNT;
	static constexpr Short ORTHO_COUNT			= Apex::ORTHO_COUNT;
	static constexpr Short ORTHO_UNITS			= Apex::ORTHO_UNITS;

#if HFSM2_SERIALIZATION_AVAILABLE()
	static constexpr Long  ACTIVE_BITS			= Apex::ACTIVE_BITS;
	static constexpr Long  RESUMABLE_BITS		= Apex::RESUMABLE_BITS;
	static constexpr Long  SERIAL_BITS			= 1 + ACTIVE_BITS + RESUMABLE_BITS;
#endif

	using Args				= ArgsT<
		Config
		, StateList
		, RegionList
		, COMPO_COUNT
		, ORTHO_COUNT
		, ORTHO_UNITS
		, ReactOrder
	HFSM2_IF_SERIALIZATION(, SERIAL_BITS)
	HFSM2_IF_PLANS(, TASK_CAPACITY)
	, Payload
	>;

	using Instance			= InstanceT<Config, Apex>;

	using ConstControl		= ConstControlT<Args>;
	using Control			= ControlT	   <Args>;
	using FullControl		= FullControlT <Args>;
	using GuardControl		= GuardControlT<Args>;
	using EventControl		= EventControlT<Args>;

	using State				= EmptyT	   <Args>;

	template <typename... TInjections>
	using StateT			= A_<TInjections...>;

#if HFSM2_LOG_INTERFACE_AVAILABLE()
	using Logger			= typename Config::LoggerInterface;
#endif

	template <typename TState>
static constexpr bool	  contains()		noexcept	{ return					contains<StateList , TState>() ;	}

	template <typename TState>
static constexpr StateID  stateId()			noexcept	{ return					   index<StateList , TState>() ;	}

	template <typename TState>
static constexpr RegionID regionId()		noexcept	{ return static_cast<RegionID>(index<RegionList, TState>());	}
};

template <typename TN, typename TA, Strategy SG, Prong NP, typename T>
struct CSubMaterialT;

template <typename TN, typename TA, Strategy SG, Prong NP, typename... TS>
struct CSubMaterialT<TN, TA, SG, NP, TL_<TS...>> final {
	using Type = CS_<TN, TA, SG, NP, TL_<TS...>>;
};

template <typename TN, typename TA, Strategy SG, Prong NP, typename... TS>
using CSubMaterial = typename CSubMaterialT<TN, TA, SG, NP, TS...>::Type;

template <typename>
struct InfoT;

template <typename TN, typename TA, typename TH>
struct InfoT<S_<TN, TA, TH>> final {
	using Type = SI_<	TH>;
};

template <typename TN, typename TA, Strategy SG, typename TH, typename... TS>
struct InfoT<C_<TN, TA, SG, TH, TS...>> final {
	using Type = CI_<	SG, TH, TS...>;
};

template <typename TN, typename TA, typename TH, typename... TS>
struct InfoT<O_<TN, TA, TH, TS...>> final {
	using Type = OI_<	TH, TS...>;
};

template <typename TN, typename TA, Strategy SG, Prong NP, typename... TS>
struct InfoT<CS_<TN, TA, SG, NP, TL_<TS...>>> final {
	using Type = CSI_<			 TL_<TS...>>;
};

template <typename T>
using Info = typename InfoT<T>::Type;

template <typename TN, typename TA, Strategy SG, Prong NP, typename T>
struct LHalfCST;

template <typename TN, typename TA, Strategy SG, Prong NP, typename... TS>
struct LHalfCST<TN, TA, SG, NP, TL_<TS...>> final {
	using Type = CS_<TN,
		TA,
		SG,
		NP,
		LHalfTypes<TS...>>;
};

template <typename TN, typename TA, Strategy SG, Prong NP, typename TL>
using LHalfCS = typename LHalfCST<TN, TA, SG, NP, TL>::Type;

template <typename TN, typename TA, Strategy SG, Prong NP, typename T>
struct RHalfCST;

template <typename TN, typename TA, Strategy SG, Prong NP, typename... TS>
struct RHalfCST<TN, TA, SG, NP, TL_<TS...>> final {
	using Indices		= TN;
	static constexpr StateID  INITIAL_ID  = Indices::STATE_ID;
	static constexpr Short	  COMPO_INDEX = Indices::COMPO_INDEX;
	static constexpr Short	  ORTHO_INDEX = Indices::ORTHO_INDEX;
	static constexpr Short	  ORTHO_UNIT  = Indices::ORTHO_UNIT;

	using LStateList	= LHalfTypes<TS...>;

	using LHalfInfo		= CSI_<LStateList>;

	using Type			= CS_<I_<INITIAL_ID  + LHalfInfo::STATE_COUNT,
		COMPO_INDEX + LHalfInfo::COMPO_COUNT,
		ORTHO_INDEX + LHalfInfo::ORTHO_COUNT,
		ORTHO_UNIT  + LHalfInfo::ORTHO_UNITS>,
	TA,
	SG,
	NP + LStateList::SIZE,
	RHalfTypes<TS...>>;
};

template <typename TN, typename TA, Strategy SG, Prong NP, typename TL>
using RHalfCS = typename RHalfCST<TN, TA, SG, NP, TL>::Type;

template <typename TN, typename TA, typename TI>
using InitialOS = MaterialT<TN, TA, TI>;

template <typename TN, typename TA, Prong NP, typename TI, typename... TR>
struct RemainingOST final {
	using Indices		= TN;
static constexpr StateID INITIAL_ID	 = Indices::STATE_ID;
static constexpr Short	 COMPO_INDEX = Indices::COMPO_INDEX;
static constexpr Short	 ORTHO_INDEX = Indices::ORTHO_INDEX;
static constexpr Short	 ORTHO_UNIT	 = Indices::ORTHO_UNIT;

	using InitialInfo	= WrapInfo<TI>;

using Type			= OS_<I_<INITIAL_ID  + InitialInfo::STATE_COUNT,
	COMPO_INDEX + InitialInfo::COMPO_COUNT,
	ORTHO_INDEX + InitialInfo::ORTHO_COUNT,
	ORTHO_UNIT  + InitialInfo::ORTHO_UNITS>,
TA,
							  NP + 1,
							  TR...>;
};

template <typename TN, typename TA, Prong NP, typename TI, typename... TR>
using RemainingOS = typename RemainingOST<TN, TA, NP, TI, TR...>::Type;

}
}

namespace hfsm2 {
	namespace detail {

		template <typename, typename>
		struct PreReactWrapperT;

		template <typename TRegion>
		struct PreReactWrapperT<TRegion, TopDown> {
			using Region		= TRegion;
			using HeadState		= typename Region::HeadState;
			using SubStates		= typename Region::SubStates;
			using EventControl	= typename Region::EventControl;

			template <typename TEvent>
			static
			HFSM2_CONSTEXPR(14)
			TaskStatus
			execute(Region& region,
			EventControl& control,
			const TEvent& event,
			const Prong active) noexcept
			{
			if (!control._consumed) {
			HeadState& headState = static_cast<HeadState&>(region);
			SubStates& subStates = static_cast<SubStates&>(region);
```
